//     PlcTask Outputs/GVL_iXlinker.EtherCAT_Master_ERxxxx.Beckhoff_ER2xxx.Beckhoff_ER2xxxEK1122.A_0046_ER2809_0021_0017.Channel_16.Output <-> Channel 16/Output
//     PlcTask Inputs/GVL_iXlinker.EtherCAT_Master_ERxxxx.Beckhoff_ER2xxx.Beckhoff_ER2xxxEK1122.A_0046_ER2809_0021_0017.WcState.WcState <-> WcState/WcState
//     PlcTask Inputs/GVL_iXlinker.EtherCAT_Master_ERxxxx.Beckhoff_ER2xxx.Beckhoff_ER2xxxEK1122.A_0046_ER2809_0021_0017.InfoData.State <-> InfoData/State
//   PLC/PLC Instance <-> EtherCAT Master ERxxxx/Beckhoff ER2xxx/Beckhoff ER2xxxEK1122/A_0047(ER2809-0021-0018)
//     PlcTask Outputs/GVL_iXlinker.EtherCAT_Master_ERxxxx.Beckhoff_ER2xxx.Beckhoff_ER2xxxEK1122.A_0047_ER2809_0021_0018.Channel_1.Output <-> Channel 1/Output
//     PlcTask Outputs/GVL_iXlinker.EtherCAT_Master_ERxxxx.Beckhoff_ER2xxx.Beckhoff_ER2xxxEK1122.A_0047_ER2809_0021_0018.Channel_2.Output <-> Channel 2/Output
//     PlcTask Outputs/GVL_iXlinker.EtherCAT_Master_ERxxxx.Beckhoff_ER2xxx.Beckhoff_ER2xxxEK1122.A_0047_ER2809_0021_0018.Channel_3.Output <-> Channel 3/Output
//     PlcTask Outputs/GVL_iXlinker.EtherCAT_Master_ERxxxx.Beckhoff_ER2xxx.Beckhoff_ER2xxxEK1122.A_0047_ER2809_0021_0018.Channel_4.Output <-> Channel 4/Output
//     PlcTask Outputs/GVL_iXlinker.EtherCAT_Master_ERxxxx.Beckhoff_ER2xxx.Beckhoff_ER2xxxEK1122.A_0047_ER2809_0021_0018.Channel_5.Output <-> Channel 5/Output
//     PlcTask Outputs/GVL_iXlinker.EtherCAT_Master_ERxxxx.Beckhoff_ER2xxx.Beckhoff_ER2xxxEK1122.A_0047_ER2809_0021_0018.Channel_6.Output <-> Channel 6/Output
//     PlcTask Outputs/GVL_iXlinker.EtherCAT_Master_ERxxxx.Beckhoff_ER2xxx.Beckhoff_ER2xxxEK1122.A_0047_ER2809_0021_0018.Channel_7.Output <-> Channel 7/Output
//     PlcTask Outputs/GVL_iXlinker.EtherCAT_Master_ERxxxx.Beckhoff_ER2xxx.Beckhoff_ER2xxxEK1122.A_0047_ER2809_0021_0018.Channel_8.Output <-> Channel 8/Output
//     PlcTask Outputs/GVL_iXlinker.EtherCAT_Master_ERxxxx.Beckhoff_ER2xxx.Beckhoff_ER2xxxEK1122.A_0047_ER2809_0021_0018.Channel_9.Output <-> Channel 9/Output
//     PlcTask Outputs/GVL_iXlinker.EtherCAT_Master_ERxxxx.Beckhoff_ER2xxx.Beckhoff_ER2xxxEK1122.A_0047_ER2809_0021_0018.Channel_10.Output <-> Channel 10/Output
//     PlcTask Outputs/GVL_iXlinker.EtherCAT_Master_ERxxxx.Beckhoff_ER2xxx.Beckhoff_ER2xxxEK1122.A_0047_ER2809_0021_0018.Channel_11.Output <-> Channel 11/Output
//     PlcTask Outputs/GVL_iXlinker.EtherCAT_Master_ERxxxx.Beckhoff_ER2xxx.Beckhoff_ER2xxxEK1122.A_0047_ER2809_0021_0018.Channel_12.Output <-> Channel 12/Output
//     PlcTask Outputs/GVL_iXlinker.EtherCAT_Master_ERxxxx.Beckhoff_ER2xxx.Beckhoff_ER2xxxEK1122.A_0047_ER2809_0021_0018.Channel_13.Output <-> Channel 13/Output
//     PlcTask Outputs/GVL_iXlinker.EtherCAT_Master_ERxxxx.Beckhoff_ER2xxx.Beckhoff_ER2xxxEK1122.A_0047_ER2809_0021_0018.Channel_14.Output <-> Channel 14/Output
//     PlcTask Outputs/GVL_iXlinker.EtherCAT_Master_ERxxxx.Beckhoff_ER2xxx.Beckhoff_ER2xxxEK1122.A_0047_ER2809_0021_0018.Channel_15.Output <-> Channel 15/Output
//     PlcTask Outputs/GVL_iXlinker.EtherCAT_Master_ERxxxx.Beckhoff_ER2xxx.Beckhoff_ER2xxxEK1122.A_0047_ER2809_0021_0018.Channel_16.Output <-> Channel 16/Output
//     PlcTask Inputs/GVL_iXlinker.EtherCAT_Master_ERxxxx.Beckhoff_ER2xxx.Beckhoff_ER2xxxEK1122.A_0047_ER2809_0021_0018.WcState.WcState <-> WcState/WcState
//     PlcTask Inputs/GVL_iXlinker.EtherCAT_Master_ERxxxx.Beckhoff_ER2xxx.Beckhoff_ER2xxxEK1122.A_0047_ER2809_0021_0018.InfoData.State <-> InfoData/State
//   PLC/PLC Instance <-> EtherCAT Master ERxxxx/Beckhoff ER2xxx/Beckhoff ER2xxxEK1122/A_0048(ER2809-0022-0016)
//     PlcTask Outputs/GVL_iXlinker.EtherCAT_Master_ERxxxx.Beckhoff_ER2xxx.Beckhoff_ER2xxxEK1122.A_0048_ER2809_0022_0016.Channel_1.Output <-> Channel 1/Output
//     PlcTask Outputs/GVL_iXlinker.EtherCAT_Master_ERxxxx.Beckhoff_ER2xxx.Beckhoff_ER2xxxEK1122.A_0048_ER2809_0022_0016.Channel_2.Output <-> Channel 2/Output
//     PlcTask Outputs/GVL_iXlinker.EtherCAT_Master_ERxxxx.Beckhoff_ER2xxx.Beckhoff_ER2xxxEK1122.A_0048_ER2809_0022_0016.Channel_3.Output <-> Channel 3/Output
//     PlcTask Outputs/GVL_iXlinker.EtherCAT_Master_ERxxxx.Beckhoff_ER2xxx.Beckhoff_ER2xxxEK1122.A_0048_ER2809_0022_0016.Channel_4.Output <-> Channel 4/Output
//     PlcTask Outputs/GVL_iXlinker.EtherCAT_Master_ERxxxx.Beckhoff_ER2xxx.Beckhoff_ER2xxxEK1122.A_0048_ER2809_0022_0016.Channel_5.Output <-> Channel 5/Output
//     PlcTask Outputs/GVL_iXlinker.EtherCAT_Master_ERxxxx.Beckhoff_ER2xxx.Beckhoff_ER2xxxEK1122.A_0048_ER2809_0022_0016.Channel_6.Output <-> Channel 6/Output
//     PlcTask Outputs/GVL_iXlinker.EtherCAT_Master_ERxxxx.Beckhoff_ER2xxx.Beckhoff_ER2xxxEK1122.A_0048_ER2809_0022_0016.Channel_7.Output <-> Channel 7/Output
//     PlcTask Outputs/GVL_iXlinker.EtherCAT_Master_ERxxxx.Beckhoff_ER2xxx.Beckhoff_ER2xxxEK1122.A_0048_ER2809_0022_0016.Channel_8.Output <-> Channel 8/Output
//     PlcTask Outputs/GVL_iXlinker.EtherCAT_Master_ERxxxx.Beckhoff_ER2xxx.Beckhoff_ER2xxxEK1122.A_0048_ER2809_0022_0016.Channel_9.Output <-> Channel 9/Output
//     PlcTask Outputs/GVL_iXlinker.EtherCAT_Master_ERxxxx.Beckhoff_ER2xxx.Beckhoff_ER2xxxEK1122.A_0048_ER2809_0022_0016.Channel_10.Output <-> Channel 10/Output
//     PlcTask Outputs/GVL_iXlinker.EtherCAT_Master_ERxxxx.Beckhoff_ER2xxx.Beckhoff_ER2xxxEK1122.A_0048_ER2809_0022_0016.Channel_11.Output <-> Channel 11/Output
//     PlcTask Outputs/GVL_iXlinker.EtherCAT_Master_ERxxxx.Beckhoff_ER2xxx.Beckhoff_ER2xxxEK1122.A_0048_ER2809_0022_0016.Channel_12.Output <-> Channel 12/Output
//     PlcTask Outputs/GVL_iXlinker.EtherCAT_Master_ERxxxx.Beckhoff_ER2xxx.Beckhoff_ER2xxxEK1122.A_0048_ER2809_0022_0016.Channel_13.Output <-> Channel 13/Output
//     PlcTask Outputs/GVL_iXlinker.EtherCAT_Master_ERxxxx.Beckhoff_ER2xxx.Beckhoff_ER2xxxEK1122.A_0048_ER2809_0022_0016.Channel_14.Output <-> Channel 14/Output
//     PlcTask Outputs/GVL_iXlinker.EtherCAT_Master_ERxxxx.Beckhoff_ER2xxx.Beckhoff_ER2xxxEK1122.A_0048_ER2809_0022_0016.Channel_15.Output <-> Channel 15/Output
//     PlcTask Outputs/GVL_iXlinker.EtherCAT_Master_ERxxxx.Beckhoff_ER2xxx.Beckhoff_ER2xxxEK1122.A_0048_ER2809_0022_0016.Channel_16.Output <-> Channel 16/Output
//     PlcTask Inputs/GVL_iXlinker.EtherCAT_Master_ERxxxx.Beckhoff_ER2xxx.Beckhoff_ER2xxxEK1122.A_0048_ER2809_0022_0016.WcState.WcState <-> WcState/WcState
//     PlcTask Inputs/GVL_iXlinker.EtherCAT_Master_ERxxxx.Beckhoff_ER2xxx.Beckhoff_ER2xxxEK1122.A_0048_ER2809_0022_0016.InfoData.State <-> InfoData/State
//   PLC/PLC Instance <-> EtherCAT Master ERxxxx/Beckhoff ER2xxx/Beckhoff ER2xxxEK1122/A_0049(ER2809-0022-0017)
//     PlcTask Outputs/GVL_iXlinker.EtherCAT_Master_ERxxxx.Beckhoff_ER2xxx.Beckhoff_ER2xxxEK1122.A_0049_ER2809_0022_0017.Channel_1.Output <-> Channel 1/Output
//     PlcTask Outputs/GVL_iXlinker.EtherCAT_Master_ERxxxx.Beckhoff_ER2xxx.Beckhoff_ER2xxxEK1122.A_0049_ER2809_0022_0017.Channel_2.Output <-> Channel 2/Output
//     PlcTask Outputs/GVL_iXlinker.EtherCAT_Master_ERxxxx.Beckhoff_ER2xxx.Beckhoff_ER2xxxEK1122.A_0049_ER2809_0022_0017.Channel_3.Output <-> Channel 3/Output
//     PlcTask Outputs/GVL_iXlinker.EtherCAT_Master_ERxxxx.Beckhoff_ER2xxx.Beckhoff_ER2xxxEK1122.A_0049_ER2809_0022_0017.Channel_4.Output <-> Channel 4/Output
//     PlcTask Outputs/GVL_iXlinker.EtherCAT_Master_ERxxxx.Beckhoff_ER2xxx.Beckhoff_ER2xxxEK1122.A_0049_ER2809_0022_0017.Channel_5.Output <-> Channel 5/Output
//     PlcTask Outputs/GVL_iXlinker.EtherCAT_Master_ERxxxx.Beckhoff_ER2xxx.Beckhoff_ER2xxxEK1122.A_0049_ER2809_0022_0017.Channel_6.Output <-> Channel 6/Output
//     PlcTask Outputs/GVL_iXlinker.EtherCAT_Master_ERxxxx.Beckhoff_ER2xxx.Beckhoff_ER2xxxEK1122.A_0049_ER2809_0022_0017.Channel_7.Output <-> Channel 7/Output
//     PlcTask Outputs/GVL_iXlinker.EtherCAT_Master_ERxxxx.Beckhoff_ER2xxx.Beckhoff_ER2xxxEK1122.A_0049_ER2809_0022_0017.Channel_8.Output <-> Channel 8/Output
//     PlcTask Outputs/GVL_iXlinker.EtherCAT_Master_ERxxxx.Beckhoff_ER2xxx.Beckhoff_ER2xxxEK1122.A_0049_ER2809_0022_0017.Channel_9.Output <-> Channel 9/Output
//     PlcTask Outputs/GVL_iXlinker.EtherCAT_Master_ERxxxx.Beckhoff_ER2xxx.Beckhoff_ER2xxxEK1122.A_0049_ER2809_0022_0017.Channel_10.Output <-> Channel 10/Output
//     PlcTask Outputs/GVL_iXlinker.EtherCAT_Master_ERxxxx.Beckhoff_ER2xxx.Beckhoff_ER2xxxEK1122.A_0049_ER2809_0022_0017.Channel_11.Output <-> Channel 11/Output
//     PlcTask Outputs/GVL_iXlinker.EtherCAT_Master_ERxxxx.Beckhoff_ER2xxx.Beckhoff_ER2xxxEK1122.A_0049_ER2809_0022_0017.Channel_12.Output <-> Channel 12/Output
//     PlcTask Outputs/GVL_iXlinker.EtherCAT_Master_ERxxxx.Beckhoff_ER2xxx.Beckhoff_ER2xxxEK1122.A_0049_ER2809_0022_0017.Channel_13.Output <-> Channel 13/Output
//     PlcTask Outputs/GVL_iXlinker.EtherCAT_Master_ERxxxx.Beckhoff_ER2xxx.Beckhoff_ER2xxxEK1122.A_0049_ER2809_0022_0017.Channel_14.Output <-> Channel 14/Output
//     PlcTask Outputs/GVL_iXlinker.EtherCAT_Master_ERxxxx.Beckhoff_ER2xxx.Beckhoff_ER2xxxEK1122.A_0049_ER2809_0022_0017.Channel_15.Output <-> Channel 15/Output
//     PlcTask Outputs/GVL_iXlinker.EtherCAT_Master_ERxxxx.Beckhoff_ER2xxx.Beckhoff_ER2xxxEK1122.A_0049_ER2809_0022_0017.Channel_16.Output <-> Channel 16/Output
//     PlcTask Inputs/GVL_iXlinker.EtherCAT_Master_ERxxxx.Beckhoff_ER2xxx.Beckhoff_ER2xxxEK1122.A_0049_ER2809_0022_0017.WcState.WcState <-> WcState/WcState
//     PlcTask Inputs/GVL_iXlinker.EtherCAT_Master_ERxxxx.Beckhoff_ER2xxx.Beckhoff_ER2xxxEK1122.A_0049_ER2809_0022_0017.InfoData.State <-> InfoData/State
//   PLC/PLC Instance <-> EtherCAT Master ERxxxx/Beckhoff ER2xxx/Beckhoff ER2xxxEK1122/A_0050(ER2809-0022-0018)
//     PlcTask Outputs/GVL_iXlinker.EtherCAT_Master_ERxxxx.Beckhoff_ER2xxx.Beckhoff_ER2xxxEK1122.A_0050_ER2809_0022_0018.Channel_1.Output <-> Channel 1/Output
//     PlcTask Outputs/GVL_iXlinker.EtherCAT_Master_ERxxxx.Beckhoff_ER2xxx.Beckhoff_ER2xxxEK1122.A_0050_ER2809_0022_0018.Channel_2.Output <-> Channel 2/Output
//     PlcTask Outputs/GVL_iXlinker.EtherCAT_Master_ERxxxx.Beckhoff_ER2xxx.Beckhoff_ER2xxxEK1122.A_0050_ER2809_0022_0018.Channel_3.Output <-> Channel 3/Output
//     PlcTask Outputs/GVL_iXlinker.EtherCAT_Master_ERxxxx.Beckhoff_ER2xxx.Beckhoff_ER2xxxEK1122.A_0050_ER2809_0022_0018.Channel_4.Output <-> Channel 4/Output
//     PlcTask Outputs/GVL_iXlinker.EtherCAT_Master_ERxxxx.Beckhoff_ER2xxx.Beckhoff_ER2xxxEK1122.A_0050_ER2809_0022_0018.Channel_5.Output <-> Channel 5/Output
//     PlcTask Outputs/GVL_iXlinker.EtherCAT_Master_ERxxxx.Beckhoff_ER2xxx.Beckhoff_ER2xxxEK1122.A_0050_ER2809_0022_0018.Channel_6.Output <-> Channel 6/Output
//     PlcTask Outputs/GVL_iXlinker.EtherCAT_Master_ERxxxx.Beckhoff_ER2xxx.Beckhoff_ER2xxxEK1122.A_0050_ER2809_0022_0018.Channel_7.Output <-> Channel 7/Output
//     PlcTask Outputs/GVL_iXlinker.EtherCAT_Master_ERxxxx.Beckhoff_ER2xxx.Beckhoff_ER2xxxEK1122.A_0050_ER2809_0022_0018.Channel_8.Output <-> Channel 8/Output
//     PlcTask Outputs/GVL_iXlinker.EtherCAT_Master_ERxxxx.Beckhoff_ER2xxx.Beckhoff_ER2xxxEK1122.A_0050_ER2809_0022_0018.Channel_9.Output <-> Channel 9/Output
//     PlcTask Outputs/GVL_iXlinker.EtherCAT_Master_ERxxxx.Beckhoff_ER2xxx.Beckhoff_ER2xxxEK1122.A_0050_ER2809_0022_0018.Channel_10.Output <-> Channel 10/Output
//     PlcTask Outputs/GVL_iXlinker.EtherCAT_Master_ERxxxx.Beckhoff_ER2xxx.Beckhoff_ER2xxxEK1122.A_0050_ER2809_0022_0018.Channel_11.Output <-> Channel 11/Output
//     PlcTask Outputs/GVL_iXlinker.EtherCAT_Master_ERxxxx.Beckhoff_ER2xxx.Beckhoff_ER2xxxEK1122.A_0050_ER2809_0022_0018.Channel_12.Output <-> Channel 12/Output
//     PlcTask Outputs/GVL_iXlinker.EtherCAT_Master_ERxxxx.Beckhoff_ER2xxx.Beckhoff_ER2xxxEK1122.A_0050_ER2809_0022_0018.Channel_13.Output <-> Channel 13/Output
//     PlcTask Outputs/GVL_iXlinker.EtherCAT_Master_ERxxxx.Beckhoff_ER2xxx.Beckhoff_ER2xxxEK1122.A_0050_ER2809_0022_0018.Channel_14.Output <-> Channel 14/Output
//     PlcTask Outputs/GVL_iXlinker.EtherCAT_Master_ERxxxx.Beckhoff_ER2xxx.Beckhoff_ER2xxxEK1122.A_0050_ER2809_0022_0018.Channel_15.Output <-> Channel 15/Output
//     PlcTask Outputs/GVL_iXlinker.EtherCAT_Master_ERxxxx.Beckhoff_ER2xxx.Beckhoff_ER2xxxEK1122.A_0050_ER2809_0022_0018.Channel_16.Output <-> Channel 16/Output
//     PlcTask Inputs/GVL_iXlinker.EtherCAT_Master_ERxxxx.Beckhoff_ER2xxx.Beckhoff_ER2xxxEK1122.A_0050_ER2809_0022_0018.WcState.WcState <-> WcState/WcState
//     PlcTask Inputs/GVL_iXlinker.EtherCAT_Master_ERxxxx.Beckhoff_ER2xxx.Beckhoff_ER2xxxEK1122.A_0050_ER2809_0022_0018.InfoData.State <-> InfoData/State
//   PLC/PLC Instance <-> EtherCAT Master ERxxxx/Beckhoff ER3xxx
//     PlcTask Inputs/GVL_iXlinker.EtherCAT_Master_ERxxxx.Beckhoff_ER3xxx.InfoData.State <-> InfoData/State
//   PLC/PLC Instance <-> EtherCAT Master ERxxxx/Beckhoff ER3xxx/Beckhoff ER3xxxEK1122
//     PlcTask Inputs/GVL_iXlinker.EtherCAT_Master_ERxxxx.Beckhoff_ER3xxx.Beckhoff_ER3xxxEK1122.InfoData.State <-> InfoData/State
//   PLC/PLC Instance <-> EtherCAT Master ERxxxx/Beckhoff ER3xxx/Beckhoff ER3xxxEK1122/Beckhoff ER3xxxsub EK1100
//     PlcTask Inputs/GVL_iXlinker.EtherCAT_Master_ERxxxx.Beckhoff_ER3xxx.Beckhoff_ER3xxxEK1122.Beckhoff_ER3xxxsub_EK1100.InfoData.State <-> InfoData/State
//   PLC/PLC Instance <-> EtherCAT Master ERxxxx/Beckhoff ER3xxx/Beckhoff ER3xxxEK1122/A_0001(ER3174-0002-0016)
//     PlcTask Inputs/GVL_iXlinker.EtherCAT_Master_ERxxxx.Beckhoff_ER3xxx.Beckhoff_ER3xxxEK1122.A_0001_ER3174_0002_0016.AI_Standard_Channel_1.Status/Underrange <-> AI Standard Channel 1/Status/Underrange
//     PlcTask Inputs/GVL_iXlinker.EtherCAT_Master_ERxxxx.Beckhoff_ER3xxx.Beckhoff_ER3xxxEK1122.A_0001_ER3174_0002_0016.AI_Standard_Channel_2.Status/Underrange <-> AI Standard Channel 2/Status/Underrange
//     PlcTask Inputs/GVL_iXlinker.EtherCAT_Master_ERxxxx.Beckhoff_ER3xxx.Beckhoff_ER3xxxEK1122.A_0001_ER3174_0002_0016.AI_Standard_Channel_3.Status/Underrange <-> AI Standard Channel 3/Status/Underrange
//     PlcTask Inputs/GVL_iXlinker.EtherCAT_Master_ERxxxx.Beckhoff_ER3xxx.Beckhoff_ER3xxxEK1122.A_0001_ER3174_0002_0016.AI_Standard_Channel_4.Status/Underrange <-> AI Standard Channel 4/Status/Underrange
//     PlcTask Inputs/GVL_iXlinker.EtherCAT_Master_ERxxxx.Beckhoff_ER3xxx.Beckhoff_ER3xxxEK1122.A_0001_ER3174_0002_0016.AI_Standard_Channel_1.Status/Overrange <-> AI Standard Channel 1/Status/Overrange
//     PlcTask Inputs/GVL_iXlinker.EtherCAT_Master_ERxxxx.Beckhoff_ER3xxx.Beckhoff_ER3xxxEK1122.A_0001_ER3174_0002_0016.AI_Standard_Channel_2.Status/Overrange <-> AI Standard Channel 2/Status/Overrange
//     PlcTask Inputs/GVL_iXlinker.EtherCAT_Master_ERxxxx.Beckhoff_ER3xxx.Beckhoff_ER3xxxEK1122.A_0001_ER3174_0002_0016.AI_Standard_Channel_3.Status/Overrange <-> AI Standard Channel 3/Status/Overrange
//     PlcTask Inputs/GVL_iXlinker.EtherCAT_Master_ERxxxx.Beckhoff_ER3xxx.Beckhoff_ER3xxxEK1122.A_0001_ER3174_0002_0016.AI_Standard_Channel_4.Status/Overrange <-> AI Standard Channel 4/Status/Overrange
//     PlcTask Inputs/GVL_iXlinker.EtherCAT_Master_ERxxxx.Beckhoff_ER3xxx.Beckhoff_ER3xxxEK1122.A_0001_ER3174_0002_0016.AI_Standard_Channel_1.Status/Limit_1 <-> AI Standard Channel 1/Status/Limit 1
//     PlcTask Inputs/GVL_iXlinker.EtherCAT_Master_ERxxxx.Beckhoff_ER3xxx.Beckhoff_ER3xxxEK1122.A_0001_ER3174_0002_0016.AI_Standard_Channel_1.Status/Limit_2 <-> AI Standard Channel 1/Status/Limit 2
//     PlcTask Inputs/GVL_iXlinker.EtherCAT_Master_ERxxxx.Beckhoff_ER3xxx.Beckhoff_ER3xxxEK1122.A_0001_ER3174_0002_0016.AI_Standard_Channel_2.Status/Limit_1 <-> AI Standard Channel 2/Status/Limit 1
//     PlcTask Inputs/GVL_iXlinker.EtherCAT_Master_ERxxxx.Beckhoff_ER3xxx.Beckhoff_ER3xxxEK1122.A_0001_ER3174_0002_0016.AI_Standard_Channel_2.Status/Limit_2 <-> AI Standard Channel 2/Status/Limit 2
//     PlcTask Inputs/GVL_iXlinker.EtherCAT_Master_ERxxxx.Beckhoff_ER3xxx.Beckhoff_ER3xxxEK1122.A_0001_ER3174_0002_0016.AI_Standard_Channel_3.Status/Limit_1 <-> AI Standard Channel 3/Status/Limit 1
//     PlcTask Inputs/GVL_iXlinker.EtherCAT_Master_ERxxxx.Beckhoff_ER3xxx.Beckhoff_ER3xxxEK1122.A_0001_ER3174_0002_0016.AI_Standard_Channel_3.Status/Limit_2 <-> AI Standard Channel 3/Status/Limit 2
//     PlcTask Inputs/GVL_iXlinker.EtherCAT_Master_ERxxxx.Beckhoff_ER3xxx.Beckhoff_ER3xxxEK1122.A_0001_ER3174_0002_0016.AI_Standard_Channel_4.Status/Limit_1 <-> AI Standard Channel 4/Status/Limit 1
//     PlcTask Inputs/GVL_iXlinker.EtherCAT_Master_ERxxxx.Beckhoff_ER3xxx.Beckhoff_ER3xxxEK1122.A_0001_ER3174_0002_0016.AI_Standard_Channel_4.Status/Limit_2 <-> AI Standard Channel 4/Status/Limit 2
//     PlcTask Inputs/GVL_iXlinker.EtherCAT_Master_ERxxxx.Beckhoff_ER3xxx.Beckhoff_ER3xxxEK1122.A_0001_ER3174_0002_0016.AI_Standard_Channel_1.Status/Error <-> AI Standard Channel 1/Status/Error
//     PlcTask Inputs/GVL_iXlinker.EtherCAT_Master_ERxxxx.Beckhoff_ER3xxx.Beckhoff_ER3xxxEK1122.A_0001_ER3174_0002_0016.AI_Standard_Channel_2.Status/Error <-> AI Standard Channel 2/Status/Error
//     PlcTask Inputs/GVL_iXlinker.EtherCAT_Master_ERxxxx.Beckhoff_ER3xxx.Beckhoff_ER3xxxEK1122.A_0001_ER3174_0002_0016.AI_Standard_Channel_3.Status/Error <-> AI Standard Channel 3/Status/Error
//     PlcTask Inputs/GVL_iXlinker.EtherCAT_Master_ERxxxx.Beckhoff_ER3xxx.Beckhoff_ER3xxxEK1122.A_0001_ER3174_0002_0016.AI_Standard_Channel_4.Status/Error <-> AI Standard Channel 4/Status/Error
//     PlcTask Inputs/GVL_iXlinker.EtherCAT_Master_ERxxxx.Beckhoff_ER3xxx.Beckhoff_ER3xxxEK1122.A_0001_ER3174_0002_0016.AI_Standard_Channel_1.Status/Sync_error <-> AI Standard Channel 1/Status/Sync error
//     PlcTask Inputs/GVL_iXlinker.EtherCAT_Master_ERxxxx.Beckhoff_ER3xxx.Beckhoff_ER3xxxEK1122.A_0001_ER3174_0002_0016.AI_Standard_Channel_2.Status/Sync_error <-> AI Standard Channel 2/Status/Sync error
//     PlcTask Inputs/GVL_iXlinker.EtherCAT_Master_ERxxxx.Beckhoff_ER3xxx.Beckhoff_ER3xxxEK1122.A_0001_ER3174_0002_0016.AI_Standard_Channel_3.Status/Sync_error <-> AI Standard Channel 3/Status/Sync error
//     PlcTask Inputs/GVL_iXlinker.EtherCAT_Master_ERxxxx.Beckhoff_ER3xxx.Beckhoff_ER3xxxEK1122.A_0001_ER3174_0002_0016.AI_Standard_Channel_4.Status/Sync_error <-> AI Standard Channel 4/Status/Sync error
//     PlcTask Inputs/GVL_iXlinker.EtherCAT_Master_ERxxxx.Beckhoff_ER3xxx.Beckhoff_ER3xxxEK1122.A_0001_ER3174_0002_0016.AI_Standard_Channel_1.Status/TxPDO_State <-> AI Standard Channel 1/Status/TxPDO State
//     PlcTask Inputs/GVL_iXlinker.EtherCAT_Master_ERxxxx.Beckhoff_ER3xxx.Beckhoff_ER3xxxEK1122.A_0001_ER3174_0002_0016.AI_Standard_Channel_2.Status/TxPDO_State <-> AI Standard Channel 2/Status/TxPDO State
//     PlcTask Inputs/GVL_iXlinker.EtherCAT_Master_ERxxxx.Beckhoff_ER3xxx.Beckhoff_ER3xxxEK1122.A_0001_ER3174_0002_0016.AI_Standard_Channel_3.Status/TxPDO_State <-> AI Standard Channel 3/Status/TxPDO State
//     PlcTask Inputs/GVL_iXlinker.EtherCAT_Master_ERxxxx.Beckhoff_ER3xxx.Beckhoff_ER3xxxEK1122.A_0001_ER3174_0002_0016.AI_Standard_Channel_4.Status/TxPDO_State <-> AI Standard Channel 4/Status/TxPDO State
//     PlcTask Inputs/GVL_iXlinker.EtherCAT_Master_ERxxxx.Beckhoff_ER3xxx.Beckhoff_ER3xxxEK1122.A_0001_ER3174_0002_0016.AI_Standard_Channel_1.Status/TxPDO_Toggle <-> AI Standard Channel 1/Status/TxPDO Toggle
//     PlcTask Inputs/GVL_iXlinker.EtherCAT_Master_ERxxxx.Beckhoff_ER3xxx.Beckhoff_ER3xxxEK1122.A_0001_ER3174_0002_0016.AI_Standard_Channel_2.Status/TxPDO_Toggle <-> AI Standard Channel 2/Status/TxPDO Toggle
//     PlcTask Inputs/GVL_iXlinker.EtherCAT_Master_ERxxxx.Beckhoff_ER3xxx.Beckhoff_ER3xxxEK1122.A_0001_ER3174_0002_0016.AI_Standard_Channel_3.Status/TxPDO_Toggle <-> AI Standard Channel 3/Status/TxPDO Toggle
//     PlcTask Inputs/GVL_iXlinker.EtherCAT_Master_ERxxxx.Beckhoff_ER3xxx.Beckhoff_ER3xxxEK1122.A_0001_ER3174_0002_0016.AI_Standard_Channel_4.Status/TxPDO_Toggle <-> AI Standard Channel 4/Status/TxPDO Toggle
//     PlcTask Inputs/GVL_iXlinker.EtherCAT_Master_ERxxxx.Beckhoff_ER3xxx.Beckhoff_ER3xxxEK1122.A_0001_ER3174_0002_0016.AI_Standard_Channel_1.Value <-> AI Standard Channel 1/Value
//     PlcTask Inputs/GVL_iXlinker.EtherCAT_Master_ERxxxx.Beckhoff_ER3xxx.Beckhoff_ER3xxxEK1122.A_0001_ER3174_0002_0016.AI_Standard_Channel_2.Value <-> AI Standard Channel 2/Value
//     PlcTask Inputs/GVL_iXlinker.EtherCAT_Master_ERxxxx.Beckhoff_ER3xxx.Beckhoff_ER3xxxEK1122.A_0001_ER3174_0002_0016.AI_Standard_Channel_3.Value <-> AI Standard Channel 3/Value
//     PlcTask Inputs/GVL_iXlinker.EtherCAT_Master_ERxxxx.Beckhoff_ER3xxx.Beckhoff_ER3xxxEK1122.A_0001_ER3174_0002_0016.AI_Standard_Channel_4.Value <-> AI Standard Channel 4/Value
//     PlcTask Inputs/GVL_iXlinker.EtherCAT_Master_ERxxxx.Beckhoff_ER3xxx.Beckhoff_ER3xxxEK1122.A_0001_ER3174_0002_0016.WcState.WcState <-> WcState/WcState
//     PlcTask Inputs/GVL_iXlinker.EtherCAT_Master_ERxxxx.Beckhoff_ER3xxx.Beckhoff_ER3xxxEK1122.A_0001_ER3174_0002_0016.WcState.InputToggle <-> WcState/InputToggle
//     PlcTask Inputs/GVL_iXlinker.EtherCAT_Master_ERxxxx.Beckhoff_ER3xxx.Beckhoff_ER3xxxEK1122.A_0001_ER3174_0002_0016.InfoData.AdsAddr <-> InfoData/AdsAddr
//     PlcTask Inputs/GVL_iXlinker.EtherCAT_Master_ERxxxx.Beckhoff_ER3xxx.Beckhoff_ER3xxxEK1122.A_0001_ER3174_0002_0016.InfoData.State <-> InfoData/State
//   PLC/PLC Instance <-> EtherCAT Master ERxxxx/Beckhoff ER3xxx/Beckhoff ER3xxxEK1122/A_0002(ER3174-0002-0022)
//     PlcTask Inputs/GVL_iXlinker.EtherCAT_Master_ERxxxx.Beckhoff_ER3xxx.Beckhoff_ER3xxxEK1122.A_0002_ER3174_0002_0022.AI_Standard_Channel_1.Status/Underrange <-> AI Standard Channel 1/Status/Underrange
//     PlcTask Inputs/GVL_iXlinker.EtherCAT_Master_ERxxxx.Beckhoff_ER3xxx.Beckhoff_ER3xxxEK1122.A_0002_ER3174_0002_0022.AI_Standard_Channel_2.Status/Underrange <-> AI Standard Channel 2/Status/Underrange
//     PlcTask Inputs/GVL_iXlinker.EtherCAT_Master_ERxxxx.Beckhoff_ER3xxx.Beckhoff_ER3xxxEK1122.A_0002_ER3174_0002_0022.AI_Standard_Channel_3.Status/Underrange <-> AI Standard Channel 3/Status/Underrange
//     PlcTask Inputs/GVL_iXlinker.EtherCAT_Master_ERxxxx.Beckhoff_ER3xxx.Beckhoff_ER3xxxEK1122.A_0002_ER3174_0002_0022.AI_Standard_Channel_4.Status/Underrange <-> AI Standard Channel 4/Status/Underrange
//     PlcTask Inputs/GVL_iXlinker.EtherCAT_Master_ERxxxx.Beckhoff_ER3xxx.Beckhoff_ER3xxxEK1122.A_0002_ER3174_0002_0022.AI_Standard_Channel_1.Status/Overrange <-> AI Standard Channel 1/Status/Overrange
//     PlcTask Inputs/GVL_iXlinker.EtherCAT_Master_ERxxxx.Beckhoff_ER3xxx.Beckhoff_ER3xxxEK1122.A_0002_ER3174_0002_0022.AI_Standard_Channel_2.Status/Overrange <-> AI Standard Channel 2/Status/Overrange
//     PlcTask Inputs/GVL_iXlinker.EtherCAT_Master_ERxxxx.Beckhoff_ER3xxx.Beckhoff_ER3xxxEK1122.A_0002_ER3174_0002_0022.AI_Standard_Channel_3.Status/Overrange <-> AI Standard Channel 3/Status/Overrange
//     PlcTask Inputs/GVL_iXlinker.EtherCAT_Master_ERxxxx.Beckhoff_ER3xxx.Beckhoff_ER3xxxEK1122.A_0002_ER3174_0002_0022.AI_Standard_Channel_4.Status/Overrange <-> AI Standard Channel 4/Status/Overrange
//     PlcTask Inputs/GVL_iXlinker.EtherCAT_Master_ERxxxx.Beckhoff_ER3xxx.Beckhoff_ER3xxxEK1122.A_0002_ER3174_0002_0022.AI_Standard_Channel_1.Status/Limit_1 <-> AI Standard Channel 1/Status/Limit 1
//     PlcTask Inputs/GVL_iXlinker.EtherCAT_Master_ERxxxx.Beckhoff_ER3xxx.Beckhoff_ER3xxxEK1122.A_0002_ER3174_0002_0022.AI_Standard_Channel_1.Status/Limit_2 <-> AI Standard Channel 1/Status/Limit 2
//     PlcTask Inputs/GVL_iXlinker.EtherCAT_Master_ERxxxx.Beckhoff_ER3xxx.Beckhoff_ER3xxxEK1122.A_0002_ER3174_0002_0022.AI_Standard_Channel_2.Status/Limit_1 <-> AI Standard Channel 2/Status/Limit 1
//     PlcTask Inputs/GVL_iXlinker.EtherCAT_Master_ERxxxx.Beckhoff_ER3xxx.Beckhoff_ER3xxxEK1122.A_0002_ER3174_0002_0022.AI_Standard_Channel_2.Status/Limit_2 <-> AI Standard Channel 2/Status/Limit 2
//     PlcTask Inputs/GVL_iXlinker.EtherCAT_Master_ERxxxx.Beckhoff_ER3xxx.Beckhoff_ER3xxxEK1122.A_0002_ER3174_0002_0022.AI_Standard_Channel_3.Status/Limit_1 <-> AI Standard Channel 3/Status/Limit 1
//     PlcTask Inputs/GVL_iXlinker.EtherCAT_Master_ERxxxx.Beckhoff_ER3xxx.Beckhoff_ER3xxxEK1122.A_0002_ER3174_0002_0022.AI_Standard_Channel_3.Status/Limit_2 <-> AI Standard Channel 3/Status/Limit 2
//     PlcTask Inputs/GVL_iXlinker.EtherCAT_Master_ERxxxx.Beckhoff_ER3xxx.Beckhoff_ER3xxxEK1122.A_0002_ER3174_0002_0022.AI_Standard_Channel_4.Status/Limit_1 <-> AI Standard Channel 4/Status/Limit 1
//     PlcTask Inputs/GVL_iXlinker.EtherCAT_Master_ERxxxx.Beckhoff_ER3xxx.Beckhoff_ER3xxxEK1122.A_0002_ER3174_0002_0022.AI_Standard_Channel_4.Status/Limit_2 <-> AI Standard Channel 4/Status/Limit 2
//     PlcTask Inputs/GVL_iXlinker.EtherCAT_Master_ERxxxx.Beckhoff_ER3xxx.Beckhoff_ER3xxxEK1122.A_0002_ER3174_0002_0022.AI_Standard_Channel_1.Status/Error <-> AI Standard Channel 1/Status/Error
//     PlcTask Inputs/GVL_iXlinker.EtherCAT_Master_ERxxxx.Beckhoff_ER3xxx.Beckhoff_ER3xxxEK1122.A_0002_ER3174_0002_0022.AI_Standard_Channel_2.Status/Error <-> AI Standard Channel 2/Status/Error
//     PlcTask Inputs/GVL_iXlinker.EtherCAT_Master_ERxxxx.Beckhoff_ER3xxx.Beckhoff_ER3xxxEK1122.A_0002_ER3174_0002_0022.AI_Standard_Channel_3.Status/Error <-> AI Standard Channel 3/Status/Error
//     PlcTask Inputs/GVL_iXlinker.EtherCAT_Master_ERxxxx.Beckhoff_ER3xxx.Beckhoff_ER3xxxEK1122.A_0002_ER3174_0002_0022.AI_Standard_Channel_4.Status/Error <-> AI Standard Channel 4/Status/Error
//     PlcTask Inputs/GVL_iXlinker.EtherCAT_Master_ERxxxx.Beckhoff_ER3xxx.Beckhoff_ER3xxxEK1122.A_0002_ER3174_0002_0022.AI_Standard_Channel_1.Status/Sync_error <-> AI Standard Channel 1/Status/Sync error
//     PlcTask Inputs/GVL_iXlinker.EtherCAT_Master_ERxxxx.Beckhoff_ER3xxx.Beckhoff_ER3xxxEK1122.A_0002_ER3174_0002_0022.AI_Standard_Channel_2.Status/Sync_error <-> AI Standard Channel 2/Status/Sync error
//     PlcTask Inputs/GVL_iXlinker.EtherCAT_Master_ERxxxx.Beckhoff_ER3xxx.Beckhoff_ER3xxxEK1122.A_0002_ER3174_0002_0022.AI_Standard_Channel_3.Status/Sync_error <-> AI Standard Channel 3/Status/Sync error
//     PlcTask Inputs/GVL_iXlinker.EtherCAT_Master_ERxxxx.Beckhoff_ER3xxx.Beckhoff_ER3xxxEK1122.A_0002_ER3174_0002_0022.AI_Standard_Channel_4.Status/Sync_error <-> AI Standard Channel 4/Status/Sync error
//     PlcTask Inputs/GVL_iXlinker.EtherCAT_Master_ERxxxx.Beckhoff_ER3xxx.Beckhoff_ER3xxxEK1122.A_0002_ER3174_0002_0022.AI_Standard_Channel_1.Status/TxPDO_State <-> AI Standard Channel 1/Status/TxPDO State
//     PlcTask Inputs/GVL_iXlinker.EtherCAT_Master_ERxxxx.Beckhoff_ER3xxx.Beckhoff_ER3xxxEK1122.A_0002_ER3174_0002_0022.AI_Standard_Channel_2.Status/TxPDO_State <-> AI Standard Channel 2/Status/TxPDO State
//     PlcTask Inputs/GVL_iXlinker.EtherCAT_Master_ERxxxx.Beckhoff_ER3xxx.Beckhoff_ER3xxxEK1122.A_0002_ER3174_0002_0022.AI_Standard_Channel_3.Status/TxPDO_State <-> AI Standard Channel 3/Status/TxPDO State
//     PlcTask Inputs/GVL_iXlinker.EtherCAT_Master_ERxxxx.Beckhoff_ER3xxx.Beckhoff_ER3xxxEK1122.A_0002_ER3174_0002_0022.AI_Standard_Channel_4.Status/TxPDO_State <-> AI Standard Channel 4/Status/TxPDO State
//     PlcTask Inputs/GVL_iXlinker.EtherCAT_Master_ERxxxx.Beckhoff_ER3xxx.Beckhoff_ER3xxxEK1122.A_0002_ER3174_0002_0022.AI_Standard_Channel_1.Status/TxPDO_Toggle <-> AI Standard Channel 1/Status/TxPDO Toggle
//     PlcTask Inputs/GVL_iXlinker.EtherCAT_Master_ERxxxx.Beckhoff_ER3xxx.Beckhoff_ER3xxxEK1122.A_0002_ER3174_0002_0022.AI_Standard_Channel_2.Status/TxPDO_Toggle <-> AI Standard Channel 2/Status/TxPDO Toggle
//     PlcTask Inputs/GVL_iXlinker.EtherCAT_Master_ERxxxx.Beckhoff_ER3xxx.Beckhoff_ER3xxxEK1122.A_0002_ER3174_0002_0022.AI_Standard_Channel_3.Status/TxPDO_Toggle <-> AI Standard Channel 3/Status/TxPDO Toggle
//     PlcTask Inputs/GVL_iXlinker.EtherCAT_Master_ERxxxx.Beckhoff_ER3xxx.Beckhoff_ER3xxxEK1122.A_0002_ER3174_0002_0022.AI_Standard_Channel_4.Status/TxPDO_Toggle <-> AI Standard Channel 4/Status/TxPDO Toggle
//     PlcTask Inputs/GVL_iXlinker.EtherCAT_Master_ERxxxx.Beckhoff_ER3xxx.Beckhoff_ER3xxxEK1122.A_0002_ER3174_0002_0022.AI_Standard_Channel_1.Value <-> AI Standard Channel 1/Value
//     PlcTask Inputs/GVL_iXlinker.EtherCAT_Master_ERxxxx.Beckhoff_ER3xxx.Beckhoff_ER3xxxEK1122.A_0002_ER3174_0002_0022.AI_Standard_Channel_2.Value <-> AI Standard Channel 2/Value
//     PlcTask Inputs/GVL_iXlinker.EtherCAT_Master_ERxxxx.Beckhoff_ER3xxx.Beckhoff_ER3xxxEK1122.A_0002_ER3174_0002_0022.AI_Standard_Channel_3.Value <-> AI Standard Channel 3/Value
//     PlcTask Inputs/GVL_iXlinker.EtherCAT_Master_ERxxxx.Beckhoff_ER3xxx.Beckhoff_ER3xxxEK1122.A_0002_ER3174_0002_0022.AI_Standard_Channel_4.Value <-> AI Standard Channel 4/Value
//     PlcTask Inputs/GVL_iXlinker.EtherCAT_Master_ERxxxx.Beckhoff_ER3xxx.Beckhoff_ER3xxxEK1122.A_0002_ER3174_0002_0022.WcState.WcState <-> WcState/WcState
//     PlcTask Inputs/GVL_iXlinker.EtherCAT_Master_ERxxxx.Beckhoff_ER3xxx.Beckhoff_ER3xxxEK1122.A_0002_ER3174_0002_0022.WcState.InputToggle <-> WcState/InputToggle
//     PlcTask Inputs/GVL_iXlinker.EtherCAT_Master_ERxxxx.Beckhoff_ER3xxx.Beckhoff_ER3xxxEK1122.A_0002_ER3174_0002_0022.InfoData.AdsAddr <-> InfoData/AdsAddr
//     PlcTask Inputs/GVL_iXlinker.EtherCAT_Master_ERxxxx.Beckhoff_ER3xxx.Beckhoff_ER3xxxEK1122.A_0002_ER3174_0002_0022.InfoData.State <-> InfoData/State
//   PLC/PLC Instance <-> EtherCAT Master ERxxxx/Beckhoff ER3xxx/Beckhoff ER3xxxEK1122/A_0003(ER3174-0002-0023)
//     PlcTask Inputs/GVL_iXlinker.EtherCAT_Master_ERxxxx.Beckhoff_ER3xxx.Beckhoff_ER3xxxEK1122.A_0003_ER3174_0002_0023.AI_Standard_Channel_1.Status/Underrange <-> AI Standard Channel 1/Status/Underrange
//     PlcTask Inputs/GVL_iXlinker.EtherCAT_Master_ERxxxx.Beckhoff_ER3xxx.Beckhoff_ER3xxxEK1122.A_0003_ER3174_0002_0023.AI_Standard_Channel_2.Status/Underrange <-> AI Standard Channel 2/Status/Underrange
//     PlcTask Inputs/GVL_iXlinker.EtherCAT_Master_ERxxxx.Beckhoff_ER3xxx.Beckhoff_ER3xxxEK1122.A_0003_ER3174_0002_0023.AI_Standard_Channel_3.Status/Underrange <-> AI Standard Channel 3/Status/Underrange
//     PlcTask Inputs/GVL_iXlinker.EtherCAT_Master_ERxxxx.Beckhoff_ER3xxx.Beckhoff_ER3xxxEK1122.A_0003_ER3174_0002_0023.AI_Standard_Channel_4.Status/Underrange <-> AI Standard Channel 4/Status/Underrange
//     PlcTask Inputs/GVL_iXlinker.EtherCAT_Master_ERxxxx.Beckhoff_ER3xxx.Beckhoff_ER3xxxEK1122.A_0003_ER3174_0002_0023.AI_Standard_Channel_1.Status/Overrange <-> AI Standard Channel 1/Status/Overrange
//     PlcTask Inputs/GVL_iXlinker.EtherCAT_Master_ERxxxx.Beckhoff_ER3xxx.Beckhoff_ER3xxxEK1122.A_0003_ER3174_0002_0023.AI_Standard_Channel_2.Status/Overrange <-> AI Standard Channel 2/Status/Overrange
//     PlcTask Inputs/GVL_iXlinker.EtherCAT_Master_ERxxxx.Beckhoff_ER3xxx.Beckhoff_ER3xxxEK1122.A_0003_ER3174_0002_0023.AI_Standard_Channel_3.Status/Overrange <-> AI Standard Channel 3/Status/Overrange
//     PlcTask Inputs/GVL_iXlinker.EtherCAT_Master_ERxxxx.Beckhoff_ER3xxx.Beckhoff_ER3xxxEK1122.A_0003_ER3174_0002_0023.AI_Standard_Channel_4.Status/Overrange <-> AI Standard Channel 4/Status/Overrange
//     PlcTask Inputs/GVL_iXlinker.EtherCAT_Master_ERxxxx.Beckhoff_ER3xxx.Beckhoff_ER3xxxEK1122.A_0003_ER3174_0002_0023.AI_Standard_Channel_1.Status/Limit_1 <-> AI Standard Channel 1/Status/Limit 1
//     PlcTask Inputs/GVL_iXlinker.EtherCAT_Master_ERxxxx.Beckhoff_ER3xxx.Beckhoff_ER3xxxEK1122.A_0003_ER3174_0002_0023.AI_Standard_Channel_1.Status/Limit_2 <-> AI Standard Channel 1/Status/Limit 2
//     PlcTask Inputs/GVL_iXlinker.EtherCAT_Master_ERxxxx.Beckhoff_ER3xxx.Beckhoff_ER3xxxEK1122.A_0003_ER3174_0002_0023.AI_Standard_Channel_2.Status/Limit_1 <-> AI Standard Channel 2/Status/Limit 1
//     PlcTask Inputs/GVL_iXlinker.EtherCAT_Master_ERxxxx.Beckhoff_ER3xxx.Beckhoff_ER3xxxEK1122.A_0003_ER3174_0002_0023.AI_Standard_Channel_2.Status/Limit_2 <-> AI Standard Channel 2/Status/Limit 2
//     PlcTask Inputs/GVL_iXlinker.EtherCAT_Master_ERxxxx.Beckhoff_ER3xxx.Beckhoff_ER3xxxEK1122.A_0003_ER3174_0002_0023.AI_Standard_Channel_3.Status/Limit_1 <-> AI Standard Channel 3/Status/Limit 1
//     PlcTask Inputs/GVL_iXlinker.EtherCAT_Master_ERxxxx.Beckhoff_ER3xxx.Beckhoff_ER3xxxEK1122.A_0003_ER3174_0002_0023.AI_Standard_Channel_3.Status/Limit_2 <-> AI Standard Channel 3/Status/Limit 2
//     PlcTask Inputs/GVL_iXlinker.EtherCAT_Master_ERxxxx.Beckhoff_ER3xxx.Beckhoff_ER3xxxEK1122.A_0003_ER3174_0002_0023.AI_Standard_Channel_4.Status/Limit_1 <-> AI Standard Channel 4/Status/Limit 1
//     PlcTask Inputs/GVL_iXlinker.EtherCAT_Master_ERxxxx.Beckhoff_ER3xxx.Beckhoff_ER3xxxEK1122.A_0003_ER3174_0002_0023.AI_Standard_Channel_4.Status/Limit_2 <-> AI Standard Channel 4/Status/Limit 2
//     PlcTask Inputs/GVL_iXlinker.EtherCAT_Master_ERxxxx.Beckhoff_ER3xxx.Beckhoff_ER3xxxEK1122.A_0003_ER3174_0002_0023.AI_Standard_Channel_1.Status/Error <-> AI Standard Channel 1/Status/Error
//     PlcTask Inputs/GVL_iXlinker.EtherCAT_Master_ERxxxx.Beckhoff_ER3xxx.Beckhoff_ER3xxxEK1122.A_0003_ER3174_0002_0023.AI_Standard_Channel_2.Status/Error <-> AI Standard Channel 2/Status/Error
//     PlcTask Inputs/GVL_iXlinker.EtherCAT_Master_ERxxxx.Beckhoff_ER3xxx.Beckhoff_ER3xxxEK1122.A_0003_ER3174_0002_0023.AI_Standard_Channel_3.Status/Error <-> AI Standard Channel 3/Status/Error
//     PlcTask Inputs/GVL_iXlinker.EtherCAT_Master_ERxxxx.Beckhoff_ER3xxx.Beckhoff_ER3xxxEK1122.A_0003_ER3174_0002_0023.AI_Standard_Channel_4.Status/Error <-> AI Standard Channel 4/Status/Error
//     PlcTask Inputs/GVL_iXlinker.EtherCAT_Master_ERxxxx.Beckhoff_ER3xxx.Beckhoff_ER3xxxEK1122.A_0003_ER3174_0002_0023.AI_Standard_Channel_1.Status/Sync_error <-> AI Standard Channel 1/Status/Sync error
//     PlcTask Inputs/GVL_iXlinker.EtherCAT_Master_ERxxxx.Beckhoff_ER3xxx.Beckhoff_ER3xxxEK1122.A_0003_ER3174_0002_0023.AI_Standard_Channel_2.Status/Sync_error <-> AI Standard Channel 2/Status/Sync error
//     PlcTask Inputs/GVL_iXlinker.EtherCAT_Master_ERxxxx.Beckhoff_ER3xxx.Beckhoff_ER3xxxEK1122.A_0003_ER3174_0002_0023.AI_Standard_Channel_3.Status/Sync_error <-> AI Standard Channel 3/Status/Sync error
//     PlcTask Inputs/GVL_iXlinker.EtherCAT_Master_ERxxxx.Beckhoff_ER3xxx.Beckhoff_ER3xxxEK1122.A_0003_ER3174_0002_0023.AI_Standard_Channel_4.Status/Sync_error <-> AI Standard Channel 4/Status/Sync error
//     PlcTask Inputs/GVL_iXlinker.EtherCAT_Master_ERxxxx.Beckhoff_ER3xxx.Beckhoff_ER3xxxEK1122.A_0003_ER3174_0002_0023.AI_Standard_Channel_1.Status/TxPDO_State <-> AI Standard Channel 1/Status/TxPDO State
//     PlcTask Inputs/GVL_iXlinker.EtherCAT_Master_ERxxxx.Beckhoff_ER3xxx.Beckhoff_ER3xxxEK1122.A_0003_ER3174_0002_0023.AI_Standard_Channel_2.Status/TxPDO_State <-> AI Standard Channel 2/Status/TxPDO State
//     PlcTask Inputs/GVL_iXlinker.EtherCAT_Master_ERxxxx.Beckhoff_ER3xxx.Beckhoff_ER3xxxEK1122.A_0003_ER3174_0002_0023.AI_Standard_Channel_3.Status/TxPDO_State <-> AI Standard Channel 3/Status/TxPDO State
//     PlcTask Inputs/GVL_iXlinker.EtherCAT_Master_ERxxxx.Beckhoff_ER3xxx.Beckhoff_ER3xxxEK1122.A_0003_ER3174_0002_0023.AI_Standard_Channel_4.Status/TxPDO_State <-> AI Standard Channel 4/Status/TxPDO State
//     PlcTask Inputs/GVL_iXlinker.EtherCAT_Master_ERxxxx.Beckhoff_ER3xxx.Beckhoff_ER3xxxEK1122.A_0003_ER3174_0002_0023.AI_Standard_Channel_1.Status/TxPDO_Toggle <-> AI Standard Channel 1/Status/TxPDO Toggle
//     PlcTask Inputs/GVL_iXlinker.EtherCAT_Master_ERxxxx.Beckhoff_ER3xxx.Beckhoff_ER3xxxEK1122.A_0003_ER3174_0002_0023.AI_Standard_Channel_2.Status/TxPDO_Toggle <-> AI Standard Channel 2/Status/TxPDO Toggle
//     PlcTask Inputs/GVL_iXlinker.EtherCAT_Master_ERxxxx.Beckhoff_ER3xxx.Beckhoff_ER3xxxEK1122.A_0003_ER3174_0002_0023.AI_Standard_Channel_3.Status/TxPDO_Toggle <-> AI Standard Channel 3/Status/TxPDO Toggle
//     PlcTask Inputs/GVL_iXlinker.EtherCAT_Master_ERxxxx.Beckhoff_ER3xxx.Beckhoff_ER3xxxEK1122.A_0003_ER3174_0002_0023.AI_Standard_Channel_4.Status/TxPDO_Toggle <-> AI Standard Channel 4/Status/TxPDO Toggle
//     PlcTask Inputs/GVL_iXlinker.EtherCAT_Master_ERxxxx.Beckhoff_ER3xxx.Beckhoff_ER3xxxEK1122.A_0003_ER3174_0002_0023.AI_Standard_Channel_1.Value <-> AI Standard Channel 1/Value
//     PlcTask Inputs/GVL_iXlinker.EtherCAT_Master_ERxxxx.Beckhoff_ER3xxx.Beckhoff_ER3xxxEK1122.A_0003_ER3174_0002_0023.AI_Standard_Channel_2.Value <-> AI Standard Channel 2/Value
//     PlcTask Inputs/GVL_iXlinker.EtherCAT_Master_ERxxxx.Beckhoff_ER3xxx.Beckhoff_ER3xxxEK1122.A_0003_ER3174_0002_0023.AI_Standard_Channel_3.Value <-> AI Standard Channel 3/Value
//     PlcTask Inputs/GVL_iXlinker.EtherCAT_Master_ERxxxx.Beckhoff_ER3xxx.Beckhoff_ER3xxxEK1122.A_0003_ER3174_0002_0023.AI_Standard_Channel_4.Value <-> AI Standard Channel 4/Value
//     PlcTask Inputs/GVL_iXlinker.EtherCAT_Master_ERxxxx.Beckhoff_ER3xxx.Beckhoff_ER3xxxEK1122.A_0003_ER3174_0002_0023.WcState.WcState <-> WcState/WcState
//     PlcTask Inputs/GVL_iXlinker.EtherCAT_Master_ERxxxx.Beckhoff_ER3xxx.Beckhoff_ER3xxxEK1122.A_0003_ER3174_0002_0023.WcState.InputToggle <-> WcState/InputToggle
//     PlcTask Inputs/GVL_iXlinker.EtherCAT_Master_ERxxxx.Beckhoff_ER3xxx.Beckhoff_ER3xxxEK1122.A_0003_ER3174_0002_0023.InfoData.AdsAddr <-> InfoData/AdsAddr
//     PlcTask Inputs/GVL_iXlinker.EtherCAT_Master_ERxxxx.Beckhoff_ER3xxx.Beckhoff_ER3xxxEK1122.A_0003_ER3174_0002_0023.InfoData.State <-> InfoData/State
//   PLC/PLC Instance <-> EtherCAT Master ERxxxx/Beckhoff ER3xxx/Beckhoff ER3xxxEK1122/A_0004(ER3184-0002-0019)
//     PlcTask Inputs/GVL_iXlinker.EtherCAT_Master_ERxxxx.Beckhoff_ER3xxx.Beckhoff_ER3xxxEK1122.A_0004_ER3184_0002_0019.AI_Standard_Channel_1.Status/Underrange <-> AI Standard Channel 1/Status/Underrange
//     PlcTask Inputs/GVL_iXlinker.EtherCAT_Master_ERxxxx.Beckhoff_ER3xxx.Beckhoff_ER3xxxEK1122.A_0004_ER3184_0002_0019.AI_Standard_Channel_2.Status/Underrange <-> AI Standard Channel 2/Status/Underrange
//     PlcTask Inputs/GVL_iXlinker.EtherCAT_Master_ERxxxx.Beckhoff_ER3xxx.Beckhoff_ER3xxxEK1122.A_0004_ER3184_0002_0019.AI_Standard_Channel_3.Status/Underrange <-> AI Standard Channel 3/Status/Underrange
//     PlcTask Inputs/GVL_iXlinker.EtherCAT_Master_ERxxxx.Beckhoff_ER3xxx.Beckhoff_ER3xxxEK1122.A_0004_ER3184_0002_0019.AI_Standard_Channel_4.Status/Underrange <-> AI Standard Channel 4/Status/Underrange
//     PlcTask Inputs/GVL_iXlinker.EtherCAT_Master_ERxxxx.Beckhoff_ER3xxx.Beckhoff_ER3xxxEK1122.A_0004_ER3184_0002_0019.AI_Standard_Channel_1.Status/Overrange <-> AI Standard Channel 1/Status/Overrange
//     PlcTask Inputs/GVL_iXlinker.EtherCAT_Master_ERxxxx.Beckhoff_ER3xxx.Beckhoff_ER3xxxEK1122.A_0004_ER3184_0002_0019.AI_Standard_Channel_2.Status/Overrange <-> AI Standard Channel 2/Status/Overrange
//     PlcTask Inputs/GVL_iXlinker.EtherCAT_Master_ERxxxx.Beckhoff_ER3xxx.Beckhoff_ER3xxxEK1122.A_0004_ER3184_0002_0019.AI_Standard_Channel_3.Status/Overrange <-> AI Standard Channel 3/Status/Overrange
//     PlcTask Inputs/GVL_iXlinker.EtherCAT_Master_ERxxxx.Beckhoff_ER3xxx.Beckhoff_ER3xxxEK1122.A_0004_ER3184_0002_0019.AI_Standard_Channel_4.Status/Overrange <-> AI Standard Channel 4/Status/Overrange
//     PlcTask Inputs/GVL_iXlinker.EtherCAT_Master_ERxxxx.Beckhoff_ER3xxx.Beckhoff_ER3xxxEK1122.A_0004_ER3184_0002_0019.AI_Standard_Channel_1.Status/Limit_1 <-> AI Standard Channel 1/Status/Limit 1
//     PlcTask Inputs/GVL_iXlinker.EtherCAT_Master_ERxxxx.Beckhoff_ER3xxx.Beckhoff_ER3xxxEK1122.A_0004_ER3184_0002_0019.AI_Standard_Channel_1.Status/Limit_2 <-> AI Standard Channel 1/Status/Limit 2
//     PlcTask Inputs/GVL_iXlinker.EtherCAT_Master_ERxxxx.Beckhoff_ER3xxx.Beckhoff_ER3xxxEK1122.A_0004_ER3184_0002_0019.AI_Standard_Channel_2.Status/Limit_1 <-> AI Standard Channel 2/Status/Limit 1
//     PlcTask Inputs/GVL_iXlinker.EtherCAT_Master_ERxxxx.Beckhoff_ER3xxx.Beckhoff_ER3xxxEK1122.A_0004_ER3184_0002_0019.AI_Standard_Channel_2.Status/Limit_2 <-> AI Standard Channel 2/Status/Limit 2
//     PlcTask Inputs/GVL_iXlinker.EtherCAT_Master_ERxxxx.Beckhoff_ER3xxx.Beckhoff_ER3xxxEK1122.A_0004_ER3184_0002_0019.AI_Standard_Channel_3.Status/Limit_1 <-> AI Standard Channel 3/Status/Limit 1
//     PlcTask Inputs/GVL_iXlinker.EtherCAT_Master_ERxxxx.Beckhoff_ER3xxx.Beckhoff_ER3xxxEK1122.A_0004_ER3184_0002_0019.AI_Standard_Channel_3.Status/Limit_2 <-> AI Standard Channel 3/Status/Limit 2
//     PlcTask Inputs/GVL_iXlinker.EtherCAT_Master_ERxxxx.Beckhoff_ER3xxx.Beckhoff_ER3xxxEK1122.A_0004_ER3184_0002_0019.AI_Standard_Channel_4.Status/Limit_1 <-> AI Standard Channel 4/Status/Limit 1
//     PlcTask Inputs/GVL_iXlinker.EtherCAT_Master_ERxxxx.Beckhoff_ER3xxx.Beckhoff_ER3xxxEK1122.A_0004_ER3184_0002_0019.AI_Standard_Channel_4.Status/Limit_2 <-> AI Standard Channel 4/Status/Limit 2
//     PlcTask Inputs/GVL_iXlinker.EtherCAT_Master_ERxxxx.Beckhoff_ER3xxx.Beckhoff_ER3xxxEK1122.A_0004_ER3184_0002_0019.AI_Standard_Channel_1.Status/Error <-> AI Standard Channel 1/Status/Error
//     PlcTask Inputs/GVL_iXlinker.EtherCAT_Master_ERxxxx.Beckhoff_ER3xxx.Beckhoff_ER3xxxEK1122.A_0004_ER3184_0002_0019.AI_Standard_Channel_2.Status/Error <-> AI Standard Channel 2/Status/Error
//     PlcTask Inputs/GVL_iXlinker.EtherCAT_Master_ERxxxx.Beckhoff_ER3xxx.Beckhoff_ER3xxxEK1122.A_0004_ER3184_0002_0019.AI_Standard_Channel_3.Status/Error <-> AI Standard Channel 3/Status/Error
//     PlcTask Inputs/GVL_iXlinker.EtherCAT_Master_ERxxxx.Beckhoff_ER3xxx.Beckhoff_ER3xxxEK1122.A_0004_ER3184_0002_0019.AI_Standard_Channel_4.Status/Error <-> AI Standard Channel 4/Status/Error
//     PlcTask Inputs/GVL_iXlinker.EtherCAT_Master_ERxxxx.Beckhoff_ER3xxx.Beckhoff_ER3xxxEK1122.A_0004_ER3184_0002_0019.AI_Standard_Channel_1.Status/Sync_error <-> AI Standard Channel 1/Status/Sync error
//     PlcTask Inputs/GVL_iXlinker.EtherCAT_Master_ERxxxx.Beckhoff_ER3xxx.Beckhoff_ER3xxxEK1122.A_0004_ER3184_0002_0019.AI_Standard_Channel_2.Status/Sync_error <-> AI Standard Channel 2/Status/Sync error
//     PlcTask Inputs/GVL_iXlinker.EtherCAT_Master_ERxxxx.Beckhoff_ER3xxx.Beckhoff_ER3xxxEK1122.A_0004_ER3184_0002_0019.AI_Standard_Channel_3.Status/Sync_error <-> AI Standard Channel 3/Status/Sync error
//     PlcTask Inputs/GVL_iXlinker.EtherCAT_Master_ERxxxx.Beckhoff_ER3xxx.Beckhoff_ER3xxxEK1122.A_0004_ER3184_0002_0019.AI_Standard_Channel_4.Status/Sync_error <-> AI Standard Channel 4/Status/Sync error
//     PlcTask Inputs/GVL_iXlinker.EtherCAT_Master_ERxxxx.Beckhoff_ER3xxx.Beckhoff_ER3xxxEK1122.A_0004_ER3184_0002_0019.AI_Standard_Channel_1.Status/TxPDO_State <-> AI Standard Channel 1/Status/TxPDO State
//     PlcTask Inputs/GVL_iXlinker.EtherCAT_Master_ERxxxx.Beckhoff_ER3xxx.Beckhoff_ER3xxxEK1122.A_0004_ER3184_0002_0019.AI_Standard_Channel_2.Status/TxPDO_State <-> AI Standard Channel 2/Status/TxPDO State
//     PlcTask Inputs/GVL_iXlinker.EtherCAT_Master_ERxxxx.Beckhoff_ER3xxx.Beckhoff_ER3xxxEK1122.A_0004_ER3184_0002_0019.AI_Standard_Channel_3.Status/TxPDO_State <-> AI Standard Channel 3/Status/TxPDO State
//     PlcTask Inputs/GVL_iXlinker.EtherCAT_Master_ERxxxx.Beckhoff_ER3xxx.Beckhoff_ER3xxxEK1122.A_0004_ER3184_0002_0019.AI_Standard_Channel_4.Status/TxPDO_State <-> AI Standard Channel 4/Status/TxPDO State
//     PlcTask Inputs/GVL_iXlinker.EtherCAT_Master_ERxxxx.Beckhoff_ER3xxx.Beckhoff_ER3xxxEK1122.A_0004_ER3184_0002_0019.AI_Standard_Channel_1.Status/TxPDO_Toggle <-> AI Standard Channel 1/Status/TxPDO Toggle
//     PlcTask Inputs/GVL_iXlinker.EtherCAT_Master_ERxxxx.Beckhoff_ER3xxx.Beckhoff_ER3xxxEK1122.A_0004_ER3184_0002_0019.AI_Standard_Channel_2.Status/TxPDO_Toggle <-> AI Standard Channel 2/Status/TxPDO Toggle
//     PlcTask Inputs/GVL_iXlinker.EtherCAT_Master_ERxxxx.Beckhoff_ER3xxx.Beckhoff_ER3xxxEK1122.A_0004_ER3184_0002_0019.AI_Standard_Channel_3.Status/TxPDO_Toggle <-> AI Standard Channel 3/Status/TxPDO Toggle
//     PlcTask Inputs/GVL_iXlinker.EtherCAT_Master_ERxxxx.Beckhoff_ER3xxx.Beckhoff_ER3xxxEK1122.A_0004_ER3184_0002_0019.AI_Standard_Channel_4.Status/TxPDO_Toggle <-> AI Standard Channel 4/Status/TxPDO Toggle
//     PlcTask Inputs/GVL_iXlinker.EtherCAT_Master_ERxxxx.Beckhoff_ER3xxx.Beckhoff_ER3xxxEK1122.A_0004_ER3184_0002_0019.AI_Standard_Channel_1.Value <-> AI Standard Channel 1/Value
//     PlcTask Inputs/GVL_iXlinker.EtherCAT_Master_ERxxxx.Beckhoff_ER3xxx.Beckhoff_ER3xxxEK1122.A_0004_ER3184_0002_0019.AI_Standard_Channel_2.Value <-> AI Standard Channel 2/Value
//     PlcTask Inputs/GVL_iXlinker.EtherCAT_Master_ERxxxx.Beckhoff_ER3xxx.Beckhoff_ER3xxxEK1122.A_0004_ER3184_0002_0019.AI_Standard_Channel_3.Value <-> AI Standard Channel 3/Value
//     PlcTask Inputs/GVL_iXlinker.EtherCAT_Master_ERxxxx.Beckhoff_ER3xxx.Beckhoff_ER3xxxEK1122.A_0004_ER3184_0002_0019.AI_Standard_Channel_4.Value <-> AI Standard Channel 4/Value
//     PlcTask Inputs/GVL_iXlinker.EtherCAT_Master_ERxxxx.Beckhoff_ER3xxx.Beckhoff_ER3xxxEK1122.A_0004_ER3184_0002_0019.WcState.WcState <-> WcState/WcState
//     PlcTask Inputs/GVL_iXlinker.EtherCAT_Master_ERxxxx.Beckhoff_ER3xxx.Beckhoff_ER3xxxEK1122.A_0004_ER3184_0002_0019.WcState.InputToggle <-> WcState/InputToggle
//     PlcTask Inputs/GVL_iXlinker.EtherCAT_Master_ERxxxx.Beckhoff_ER3xxx.Beckhoff_ER3xxxEK1122.A_0004_ER3184_0002_0019.InfoData.AdsAddr <-> InfoData/AdsAddr
//     PlcTask Inputs/GVL_iXlinker.EtherCAT_Master_ERxxxx.Beckhoff_ER3xxx.Beckhoff_ER3xxxEK1122.A_0004_ER3184_0002_0019.InfoData.State <-> InfoData/State
//   PLC/PLC Instance <-> EtherCAT Master ERxxxx/Beckhoff ER3xxx/Beckhoff ER3xxxEK1122/A_0005(ER3184-0002-0020)
//     PlcTask Inputs/GVL_iXlinker.EtherCAT_Master_ERxxxx.Beckhoff_ER3xxx.Beckhoff_ER3xxxEK1122.A_0005_ER3184_0002_0020.AI_Standard_Channel_1.Status/Underrange <-> AI Standard Channel 1/Status/Underrange
//     PlcTask Inputs/GVL_iXlinker.EtherCAT_Master_ERxxxx.Beckhoff_ER3xxx.Beckhoff_ER3xxxEK1122.A_0005_ER3184_0002_0020.AI_Standard_Channel_2.Status/Underrange <-> AI Standard Channel 2/Status/Underrange
//     PlcTask Inputs/GVL_iXlinker.EtherCAT_Master_ERxxxx.Beckhoff_ER3xxx.Beckhoff_ER3xxxEK1122.A_0005_ER3184_0002_0020.AI_Standard_Channel_3.Status/Underrange <-> AI Standard Channel 3/Status/Underrange
//     PlcTask Inputs/GVL_iXlinker.EtherCAT_Master_ERxxxx.Beckhoff_ER3xxx.Beckhoff_ER3xxxEK1122.A_0005_ER3184_0002_0020.AI_Standard_Channel_4.Status/Underrange <-> AI Standard Channel 4/Status/Underrange
//     PlcTask Inputs/GVL_iXlinker.EtherCAT_Master_ERxxxx.Beckhoff_ER3xxx.Beckhoff_ER3xxxEK1122.A_0005_ER3184_0002_0020.AI_Standard_Channel_1.Status/Overrange <-> AI Standard Channel 1/Status/Overrange
//     PlcTask Inputs/GVL_iXlinker.EtherCAT_Master_ERxxxx.Beckhoff_ER3xxx.Beckhoff_ER3xxxEK1122.A_0005_ER3184_0002_0020.AI_Standard_Channel_2.Status/Overrange <-> AI Standard Channel 2/Status/Overrange
//     PlcTask Inputs/GVL_iXlinker.EtherCAT_Master_ERxxxx.Beckhoff_ER3xxx.Beckhoff_ER3xxxEK1122.A_0005_ER3184_0002_0020.AI_Standard_Channel_3.Status/Overrange <-> AI Standard Channel 3/Status/Overrange
//     PlcTask Inputs/GVL_iXlinker.EtherCAT_Master_ERxxxx.Beckhoff_ER3xxx.Beckhoff_ER3xxxEK1122.A_0005_ER3184_0002_0020.AI_Standard_Channel_4.Status/Overrange <-> AI Standard Channel 4/Status/Overrange
//     PlcTask Inputs/GVL_iXlinker.EtherCAT_Master_ERxxxx.Beckhoff_ER3xxx.Beckhoff_ER3xxxEK1122.A_0005_ER3184_0002_0020.AI_Standard_Channel_1.Status/Limit_1 <-> AI Standard Channel 1/Status/Limit 1
//     PlcTask Inputs/GVL_iXlinker.EtherCAT_Master_ERxxxx.Beckhoff_ER3xxx.Beckhoff_ER3xxxEK1122.A_0005_ER3184_0002_0020.AI_Standard_Channel_1.Status/Limit_2 <-> AI Standard Channel 1/Status/Limit 2
//     PlcTask Inputs/GVL_iXlinker.EtherCAT_Master_ERxxxx.Beckhoff_ER3xxx.Beckhoff_ER3xxxEK1122.A_0005_ER3184_0002_0020.AI_Standard_Channel_2.Status/Limit_1 <-> AI Standard Channel 2/Status/Limit 1
//     PlcTask Inputs/GVL_iXlinker.EtherCAT_Master_ERxxxx.Beckhoff_ER3xxx.Beckhoff_ER3xxxEK1122.A_0005_ER3184_0002_0020.AI_Standard_Channel_2.Status/Limit_2 <-> AI Standard Channel 2/Status/Limit 2
//     PlcTask Inputs/GVL_iXlinker.EtherCAT_Master_ERxxxx.Beckhoff_ER3xxx.Beckhoff_ER3xxxEK1122.A_0005_ER3184_0002_0020.AI_Standard_Channel_3.Status/Limit_1 <-> AI Standard Channel 3/Status/Limit 1
//     PlcTask Inputs/GVL_iXlinker.EtherCAT_Master_ERxxxx.Beckhoff_ER3xxx.Beckhoff_ER3xxxEK1122.A_0005_ER3184_0002_0020.AI_Standard_Channel_3.Status/Limit_2 <-> AI Standard Channel 3/Status/Limit 2
//     PlcTask Inputs/GVL_iXlinker.EtherCAT_Master_ERxxxx.Beckhoff_ER3xxx.Beckhoff_ER3xxxEK1122.A_0005_ER3184_0002_0020.AI_Standard_Channel_4.Status/Limit_1 <-> AI Standard Channel 4/Status/Limit 1
//     PlcTask Inputs/GVL_iXlinker.EtherCAT_Master_ERxxxx.Beckhoff_ER3xxx.Beckhoff_ER3xxxEK1122.A_0005_ER3184_0002_0020.AI_Standard_Channel_4.Status/Limit_2 <-> AI Standard Channel 4/Status/Limit 2
//     PlcTask Inputs/GVL_iXlinker.EtherCAT_Master_ERxxxx.Beckhoff_ER3xxx.Beckhoff_ER3xxxEK1122.A_0005_ER3184_0002_0020.AI_Standard_Channel_1.Status/Error <-> AI Standard Channel 1/Status/Error
//     PlcTask Inputs/GVL_iXlinker.EtherCAT_Master_ERxxxx.Beckhoff_ER3xxx.Beckhoff_ER3xxxEK1122.A_0005_ER3184_0002_0020.AI_Standard_Channel_2.Status/Error <-> AI Standard Channel 2/Status/Error
//     PlcTask Inputs/GVL_iXlinker.EtherCAT_Master_ERxxxx.Beckhoff_ER3xxx.Beckhoff_ER3xxxEK1122.A_0005_ER3184_0002_0020.AI_Standard_Channel_3.Status/Error <-> AI Standard Channel 3/Status/Error
//     PlcTask Inputs/GVL_iXlinker.EtherCAT_Master_ERxxxx.Beckhoff_ER3xxx.Beckhoff_ER3xxxEK1122.A_0005_ER3184_0002_0020.AI_Standard_Channel_4.Status/Error <-> AI Standard Channel 4/Status/Error
//     PlcTask Inputs/GVL_iXlinker.EtherCAT_Master_ERxxxx.Beckhoff_ER3xxx.Beckhoff_ER3xxxEK1122.A_0005_ER3184_0002_0020.AI_Standard_Channel_1.Status/Sync_error <-> AI Standard Channel 1/Status/Sync error
//     PlcTask Inputs/GVL_iXlinker.EtherCAT_Master_ERxxxx.Beckhoff_ER3xxx.Beckhoff_ER3xxxEK1122.A_0005_ER3184_0002_0020.AI_Standard_Channel_2.Status/Sync_error <-> AI Standard Channel 2/Status/Sync error
//     PlcTask Inputs/GVL_iXlinker.EtherCAT_Master_ERxxxx.Beckhoff_ER3xxx.Beckhoff_ER3xxxEK1122.A_0005_ER3184_0002_0020.AI_Standard_Channel_3.Status/Sync_error <-> AI Standard Channel 3/Status/Sync error
//     PlcTask Inputs/GVL_iXlinker.EtherCAT_Master_ERxxxx.Beckhoff_ER3xxx.Beckhoff_ER3xxxEK1122.A_0005_ER3184_0002_0020.AI_Standard_Channel_4.Status/Sync_error <-> AI Standard Channel 4/Status/Sync error
//     PlcTask Inputs/GVL_iXlinker.EtherCAT_Master_ERxxxx.Beckhoff_ER3xxx.Beckhoff_ER3xxxEK1122.A_0005_ER3184_0002_0020.AI_Standard_Channel_1.Status/TxPDO_State <-> AI Standard Channel 1/Status/TxPDO State
//     PlcTask Inputs/GVL_iXlinker.EtherCAT_Master_ERxxxx.Beckhoff_ER3xxx.Beckhoff_ER3xxxEK1122.A_0005_ER3184_0002_0020.AI_Standard_Channel_2.Status/TxPDO_State <-> AI Standard Channel 2/Status/TxPDO State
//     PlcTask Inputs/GVL_iXlinker.EtherCAT_Master_ERxxxx.Beckhoff_ER3xxx.Beckhoff_ER3xxxEK1122.A_0005_ER3184_0002_0020.AI_Standard_Channel_3.Status/TxPDO_State <-> AI Standard Channel 3/Status/TxPDO State
//     PlcTask Inputs/GVL_iXlinker.EtherCAT_Master_ERxxxx.Beckhoff_ER3xxx.Beckhoff_ER3xxxEK1122.A_0005_ER3184_0002_0020.AI_Standard_Channel_4.Status/TxPDO_State <-> AI Standard Channel 4/Status/TxPDO State
//     PlcTask Inputs/GVL_iXlinker.EtherCAT_Master_ERxxxx.Beckhoff_ER3xxx.Beckhoff_ER3xxxEK1122.A_0005_ER3184_0002_0020.AI_Standard_Channel_1.Status/TxPDO_Toggle <-> AI Standard Channel 1/Status/TxPDO Toggle
//     PlcTask Inputs/GVL_iXlinker.EtherCAT_Master_ERxxxx.Beckhoff_ER3xxx.Beckhoff_ER3xxxEK1122.A_0005_ER3184_0002_0020.AI_Standard_Channel_2.Status/TxPDO_Toggle <-> AI Standard Channel 2/Status/TxPDO Toggle
//     PlcTask Inputs/GVL_iXlinker.EtherCAT_Master_ERxxxx.Beckhoff_ER3xxx.Beckhoff_ER3xxxEK1122.A_0005_ER3184_0002_0020.AI_Standard_Channel_3.Status/TxPDO_Toggle <-> AI Standard Channel 3/Status/TxPDO Toggle
//     PlcTask Inputs/GVL_iXlinker.EtherCAT_Master_ERxxxx.Beckhoff_ER3xxx.Beckhoff_ER3xxxEK1122.A_0005_ER3184_0002_0020.AI_Standard_Channel_4.Status/TxPDO_Toggle <-> AI Standard Channel 4/Status/TxPDO Toggle
//     PlcTask Inputs/GVL_iXlinker.EtherCAT_Master_ERxxxx.Beckhoff_ER3xxx.Beckhoff_ER3xxxEK1122.A_0005_ER3184_0002_0020.AI_Standard_Channel_1.Value <-> AI Standard Channel 1/Value
//     PlcTask Inputs/GVL_iXlinker.EtherCAT_Master_ERxxxx.Beckhoff_ER3xxx.Beckhoff_ER3xxxEK1122.A_0005_ER3184_0002_0020.AI_Standard_Channel_2.Value <-> AI Standard Channel 2/Value
//     PlcTask Inputs/GVL_iXlinker.EtherCAT_Master_ERxxxx.Beckhoff_ER3xxx.Beckhoff_ER3xxxEK1122.A_0005_ER3184_0002_0020.AI_Standard_Channel_3.Value <-> AI Standard Channel 3/Value
//     PlcTask Inputs/GVL_iXlinker.EtherCAT_Master_ERxxxx.Beckhoff_ER3xxx.Beckhoff_ER3xxxEK1122.A_0005_ER3184_0002_0020.AI_Standard_Channel_4.Value <-> AI Standard Channel 4/Value
//     PlcTask Inputs/GVL_iXlinker.EtherCAT_Master_ERxxxx.Beckhoff_ER3xxx.Beckhoff_ER3xxxEK1122.A_0005_ER3184_0002_0020.WcState.WcState <-> WcState/WcState
//     PlcTask Inputs/GVL_iXlinker.EtherCAT_Master_ERxxxx.Beckhoff_ER3xxx.Beckhoff_ER3xxxEK1122.A_0005_ER3184_0002_0020.WcState.InputToggle <-> WcState/InputToggle
//     PlcTask Inputs/GVL_iXlinker.EtherCAT_Master_ERxxxx.Beckhoff_ER3xxx.Beckhoff_ER3xxxEK1122.A_0005_ER3184_0002_0020.InfoData.AdsAddr <-> InfoData/AdsAddr
//     PlcTask Inputs/GVL_iXlinker.EtherCAT_Master_ERxxxx.Beckhoff_ER3xxx.Beckhoff_ER3xxxEK1122.A_0005_ER3184_0002_0020.InfoData.State <-> InfoData/State
//   PLC/PLC Instance <-> EtherCAT Master ERxxxx/Beckhoff ER3xxx/Beckhoff ER3xxxEK1122/A_0006(ER3184-0002-0021)
//     PlcTask Inputs/GVL_iXlinker.EtherCAT_Master_ERxxxx.Beckhoff_ER3xxx.Beckhoff_ER3xxxEK1122.A_0006_ER3184_0002_0021.AI_Standard_Channel_1.Status/Underrange <-> AI Standard Channel 1/Status/Underrange
//     PlcTask Inputs/GVL_iXlinker.EtherCAT_Master_ERxxxx.Beckhoff_ER3xxx.Beckhoff_ER3xxxEK1122.A_0006_ER3184_0002_0021.AI_Standard_Channel_2.Status/Underrange <-> AI Standard Channel 2/Status/Underrange
//     PlcTask Inputs/GVL_iXlinker.EtherCAT_Master_ERxxxx.Beckhoff_ER3xxx.Beckhoff_ER3xxxEK1122.A_0006_ER3184_0002_0021.AI_Standard_Channel_3.Status/Underrange <-> AI Standard Channel 3/Status/Underrange
//     PlcTask Inputs/GVL_iXlinker.EtherCAT_Master_ERxxxx.Beckhoff_ER3xxx.Beckhoff_ER3xxxEK1122.A_0006_ER3184_0002_0021.AI_Standard_Channel_4.Status/Underrange <-> AI Standard Channel 4/Status/Underrange
//     PlcTask Inputs/GVL_iXlinker.EtherCAT_Master_ERxxxx.Beckhoff_ER3xxx.Beckhoff_ER3xxxEK1122.A_0006_ER3184_0002_0021.AI_Standard_Channel_1.Status/Overrange <-> AI Standard Channel 1/Status/Overrange
//     PlcTask Inputs/GVL_iXlinker.EtherCAT_Master_ERxxxx.Beckhoff_ER3xxx.Beckhoff_ER3xxxEK1122.A_0006_ER3184_0002_0021.AI_Standard_Channel_2.Status/Overrange <-> AI Standard Channel 2/Status/Overrange
//     PlcTask Inputs/GVL_iXlinker.EtherCAT_Master_ERxxxx.Beckhoff_ER3xxx.Beckhoff_ER3xxxEK1122.A_0006_ER3184_0002_0021.AI_Standard_Channel_3.Status/Overrange <-> AI Standard Channel 3/Status/Overrange
//     PlcTask Inputs/GVL_iXlinker.EtherCAT_Master_ERxxxx.Beckhoff_ER3xxx.Beckhoff_ER3xxxEK1122.A_0006_ER3184_0002_0021.AI_Standard_Channel_4.Status/Overrange <-> AI Standard Channel 4/Status/Overrange
//     PlcTask Inputs/GVL_iXlinker.EtherCAT_Master_ERxxxx.Beckhoff_ER3xxx.Beckhoff_ER3xxxEK1122.A_0006_ER3184_0002_0021.AI_Standard_Channel_1.Status/Limit_1 <-> AI Standard Channel 1/Status/Limit 1
//     PlcTask Inputs/GVL_iXlinker.EtherCAT_Master_ERxxxx.Beckhoff_ER3xxx.Beckhoff_ER3xxxEK1122.A_0006_ER3184_0002_0021.AI_Standard_Channel_1.Status/Limit_2 <-> AI Standard Channel 1/Status/Limit 2
//     PlcTask Inputs/GVL_iXlinker.EtherCAT_Master_ERxxxx.Beckhoff_ER3xxx.Beckhoff_ER3xxxEK1122.A_0006_ER3184_0002_0021.AI_Standard_Channel_2.Status/Limit_1 <-> AI Standard Channel 2/Status/Limit 1
//     PlcTask Inputs/GVL_iXlinker.EtherCAT_Master_ERxxxx.Beckhoff_ER3xxx.Beckhoff_ER3xxxEK1122.A_0006_ER3184_0002_0021.AI_Standard_Channel_2.Status/Limit_2 <-> AI Standard Channel 2/Status/Limit 2
//     PlcTask Inputs/GVL_iXlinker.EtherCAT_Master_ERxxxx.Beckhoff_ER3xxx.Beckhoff_ER3xxxEK1122.A_0006_ER3184_0002_0021.AI_Standard_Channel_3.Status/Limit_1 <-> AI Standard Channel 3/Status/Limit 1
//     PlcTask Inputs/GVL_iXlinker.EtherCAT_Master_ERxxxx.Beckhoff_ER3xxx.Beckhoff_ER3xxxEK1122.A_0006_ER3184_0002_0021.AI_Standard_Channel_3.Status/Limit_2 <-> AI Standard Channel 3/Status/Limit 2
//     PlcTask Inputs/GVL_iXlinker.EtherCAT_Master_ERxxxx.Beckhoff_ER3xxx.Beckhoff_ER3xxxEK1122.A_0006_ER3184_0002_0021.AI_Standard_Channel_4.Status/Limit_1 <-> AI Standard Channel 4/Status/Limit 1
//     PlcTask Inputs/GVL_iXlinker.EtherCAT_Master_ERxxxx.Beckhoff_ER3xxx.Beckhoff_ER3xxxEK1122.A_0006_ER3184_0002_0021.AI_Standard_Channel_4.Status/Limit_2 <-> AI Standard Channel 4/Status/Limit 2
//     PlcTask Inputs/GVL_iXlinker.EtherCAT_Master_ERxxxx.Beckhoff_ER3xxx.Beckhoff_ER3xxxEK1122.A_0006_ER3184_0002_0021.AI_Standard_Channel_1.Status/Error <-> AI Standard Channel 1/Status/Error
//     PlcTask Inputs/GVL_iXlinker.EtherCAT_Master_ERxxxx.Beckhoff_ER3xxx.Beckhoff_ER3xxxEK1122.A_0006_ER3184_0002_0021.AI_Standard_Channel_2.Status/Error <-> AI Standard Channel 2/Status/Error
//     PlcTask Inputs/GVL_iXlinker.EtherCAT_Master_ERxxxx.Beckhoff_ER3xxx.Beckhoff_ER3xxxEK1122.A_0006_ER3184_0002_0021.AI_Standard_Channel_3.Status/Error <-> AI Standard Channel 3/Status/Error
//     PlcTask Inputs/GVL_iXlinker.EtherCAT_Master_ERxxxx.Beckhoff_ER3xxx.Beckhoff_ER3xxxEK1122.A_0006_ER3184_0002_0021.AI_Standard_Channel_4.Status/Error <-> AI Standard Channel 4/Status/Error
//     PlcTask Inputs/GVL_iXlinker.EtherCAT_Master_ERxxxx.Beckhoff_ER3xxx.Beckhoff_ER3xxxEK1122.A_0006_ER3184_0002_0021.AI_Standard_Channel_1.Status/Sync_error <-> AI Standard Channel 1/Status/Sync error
//     PlcTask Inputs/GVL_iXlinker.EtherCAT_Master_ERxxxx.Beckhoff_ER3xxx.Beckhoff_ER3xxxEK1122.A_0006_ER3184_0002_0021.AI_Standard_Channel_2.Status/Sync_error <-> AI Standard Channel 2/Status/Sync error
//     PlcTask Inputs/GVL_iXlinker.EtherCAT_Master_ERxxxx.Beckhoff_ER3xxx.Beckhoff_ER3xxxEK1122.A_0006_ER3184_0002_0021.AI_Standard_Channel_3.Status/Sync_error <-> AI Standard Channel 3/Status/Sync error
//     PlcTask Inputs/GVL_iXlinker.EtherCAT_Master_ERxxxx.Beckhoff_ER3xxx.Beckhoff_ER3xxxEK1122.A_0006_ER3184_0002_0021.AI_Standard_Channel_4.Status/Sync_error <-> AI Standard Channel 4/Status/Sync error
//     PlcTask Inputs/GVL_iXlinker.EtherCAT_Master_ERxxxx.Beckhoff_ER3xxx.Beckhoff_ER3xxxEK1122.A_0006_ER3184_0002_0021.AI_Standard_Channel_1.Status/TxPDO_State <-> AI Standard Channel 1/Status/TxPDO State
//     PlcTask Inputs/GVL_iXlinker.EtherCAT_Master_ERxxxx.Beckhoff_ER3xxx.Beckhoff_ER3xxxEK1122.A_0006_ER3184_0002_0021.AI_Standard_Channel_2.Status/TxPDO_State <-> AI Standard Channel 2/Status/TxPDO State
//     PlcTask Inputs/GVL_iXlinker.EtherCAT_Master_ERxxxx.Beckhoff_ER3xxx.Beckhoff_ER3xxxEK1122.A_0006_ER3184_0002_0021.AI_Standard_Channel_3.Status/TxPDO_State <-> AI Standard Channel 3/Status/TxPDO State
//     PlcTask Inputs/GVL_iXlinker.EtherCAT_Master_ERxxxx.Beckhoff_ER3xxx.Beckhoff_ER3xxxEK1122.A_0006_ER3184_0002_0021.AI_Standard_Channel_4.Status/TxPDO_State <-> AI Standard Channel 4/Status/TxPDO State
//     PlcTask Inputs/GVL_iXlinker.EtherCAT_Master_ERxxxx.Beckhoff_ER3xxx.Beckhoff_ER3xxxEK1122.A_0006_ER3184_0002_0021.AI_Standard_Channel_1.Status/TxPDO_Toggle <-> AI Standard Channel 1/Status/TxPDO Toggle
//     PlcTask Inputs/GVL_iXlinker.EtherCAT_Master_ERxxxx.Beckhoff_ER3xxx.Beckhoff_ER3xxxEK1122.A_0006_ER3184_0002_0021.AI_Standard_Channel_2.Status/TxPDO_Toggle <-> AI Standard Channel 2/Status/TxPDO Toggle
//     PlcTask Inputs/GVL_iXlinker.EtherCAT_Master_ERxxxx.Beckhoff_ER3xxx.Beckhoff_ER3xxxEK1122.A_0006_ER3184_0002_0021.AI_Standard_Channel_3.Status/TxPDO_Toggle <-> AI Standard Channel 3/Status/TxPDO Toggle
//     PlcTask Inputs/GVL_iXlinker.EtherCAT_Master_ERxxxx.Beckhoff_ER3xxx.Beckhoff_ER3xxxEK1122.A_0006_ER3184_0002_0021.AI_Standard_Channel_4.Status/TxPDO_Toggle <-> AI Standard Channel 4/Status/TxPDO Toggle
//     PlcTask Inputs/GVL_iXlinker.EtherCAT_Master_ERxxxx.Beckhoff_ER3xxx.Beckhoff_ER3xxxEK1122.A_0006_ER3184_0002_0021.AI_Standard_Channel_1.Value <-> AI Standard Channel 1/Value
//     PlcTask Inputs/GVL_iXlinker.EtherCAT_Master_ERxxxx.Beckhoff_ER3xxx.Beckhoff_ER3xxxEK1122.A_0006_ER3184_0002_0021.AI_Standard_Channel_2.Value <-> AI Standard Channel 2/Value
//     PlcTask Inputs/GVL_iXlinker.EtherCAT_Master_ERxxxx.Beckhoff_ER3xxx.Beckhoff_ER3xxxEK1122.A_0006_ER3184_0002_0021.AI_Standard_Channel_3.Value <-> AI Standard Channel 3/Value
//     PlcTask Inputs/GVL_iXlinker.EtherCAT_Master_ERxxxx.Beckhoff_ER3xxx.Beckhoff_ER3xxxEK1122.A_0006_ER3184_0002_0021.AI_Standard_Channel_4.Value <-> AI Standard Channel 4/Value
//     PlcTask Inputs/GVL_iXlinker.EtherCAT_Master_ERxxxx.Beckhoff_ER3xxx.Beckhoff_ER3xxxEK1122.A_0006_ER3184_0002_0021.WcState.WcState <-> WcState/WcState
//     PlcTask Inputs/GVL_iXlinker.EtherCAT_Master_ERxxxx.Beckhoff_ER3xxx.Beckhoff_ER3xxxEK1122.A_0006_ER3184_0002_0021.WcState.InputToggle <-> WcState/InputToggle
//     PlcTask Inputs/GVL_iXlinker.EtherCAT_Master_ERxxxx.Beckhoff_ER3xxx.Beckhoff_ER3xxxEK1122.A_0006_ER3184_0002_0021.InfoData.AdsAddr <-> InfoData/AdsAddr
//     PlcTask Inputs/GVL_iXlinker.EtherCAT_Master_ERxxxx.Beckhoff_ER3xxx.Beckhoff_ER3xxxEK1122.A_0006_ER3184_0002_0021.InfoData.State <-> InfoData/State
//   PLC/PLC Instance <-> EtherCAT Master ERxxxx/Beckhoff ER3xxx/Beckhoff ER3xxxEK1122/A_0007(ER3184-1002-0020)
//     PlcTask Inputs/GVL_iXlinker.EtherCAT_Master_ERxxxx.Beckhoff_ER3xxx.Beckhoff_ER3xxxEK1122.A_0007_ER3184_1002_0020.AI_Standard_Channel_1.Status/Underrange <-> AI Standard Channel 1/Status/Underrange
//     PlcTask Inputs/GVL_iXlinker.EtherCAT_Master_ERxxxx.Beckhoff_ER3xxx.Beckhoff_ER3xxxEK1122.A_0007_ER3184_1002_0020.AI_Standard_Channel_2.Status/Underrange <-> AI Standard Channel 2/Status/Underrange
//     PlcTask Inputs/GVL_iXlinker.EtherCAT_Master_ERxxxx.Beckhoff_ER3xxx.Beckhoff_ER3xxxEK1122.A_0007_ER3184_1002_0020.AI_Standard_Channel_3.Status/Underrange <-> AI Standard Channel 3/Status/Underrange
//     PlcTask Inputs/GVL_iXlinker.EtherCAT_Master_ERxxxx.Beckhoff_ER3xxx.Beckhoff_ER3xxxEK1122.A_0007_ER3184_1002_0020.AI_Standard_Channel_4.Status/Underrange <-> AI Standard Channel 4/Status/Underrange
//     PlcTask Inputs/GVL_iXlinker.EtherCAT_Master_ERxxxx.Beckhoff_ER3xxx.Beckhoff_ER3xxxEK1122.A_0007_ER3184_1002_0020.AI_Standard_Channel_1.Status/Overrange <-> AI Standard Channel 1/Status/Overrange
//     PlcTask Inputs/GVL_iXlinker.EtherCAT_Master_ERxxxx.Beckhoff_ER3xxx.Beckhoff_ER3xxxEK1122.A_0007_ER3184_1002_0020.AI_Standard_Channel_2.Status/Overrange <-> AI Standard Channel 2/Status/Overrange
//     PlcTask Inputs/GVL_iXlinker.EtherCAT_Master_ERxxxx.Beckhoff_ER3xxx.Beckhoff_ER3xxxEK1122.A_0007_ER3184_1002_0020.AI_Standard_Channel_3.Status/Overrange <-> AI Standard Channel 3/Status/Overrange
//     PlcTask Inputs/GVL_iXlinker.EtherCAT_Master_ERxxxx.Beckhoff_ER3xxx.Beckhoff_ER3xxxEK1122.A_0007_ER3184_1002_0020.AI_Standard_Channel_4.Status/Overrange <-> AI Standard Channel 4/Status/Overrange
//     PlcTask Inputs/GVL_iXlinker.EtherCAT_Master_ERxxxx.Beckhoff_ER3xxx.Beckhoff_ER3xxxEK1122.A_0007_ER3184_1002_0020.AI_Standard_Channel_1.Status/Limit_1 <-> AI Standard Channel 1/Status/Limit 1
//     PlcTask Inputs/GVL_iXlinker.EtherCAT_Master_ERxxxx.Beckhoff_ER3xxx.Beckhoff_ER3xxxEK1122.A_0007_ER3184_1002_0020.AI_Standard_Channel_1.Status/Limit_2 <-> AI Standard Channel 1/Status/Limit 2
//     PlcTask Inputs/GVL_iXlinker.EtherCAT_Master_ERxxxx.Beckhoff_ER3xxx.Beckhoff_ER3xxxEK1122.A_0007_ER3184_1002_0020.AI_Standard_Channel_2.Status/Limit_1 <-> AI Standard Channel 2/Status/Limit 1
//     PlcTask Inputs/GVL_iXlinker.EtherCAT_Master_ERxxxx.Beckhoff_ER3xxx.Beckhoff_ER3xxxEK1122.A_0007_ER3184_1002_0020.AI_Standard_Channel_2.Status/Limit_2 <-> AI Standard Channel 2/Status/Limit 2
//     PlcTask Inputs/GVL_iXlinker.EtherCAT_Master_ERxxxx.Beckhoff_ER3xxx.Beckhoff_ER3xxxEK1122.A_0007_ER3184_1002_0020.AI_Standard_Channel_3.Status/Limit_1 <-> AI Standard Channel 3/Status/Limit 1
//     PlcTask Inputs/GVL_iXlinker.EtherCAT_Master_ERxxxx.Beckhoff_ER3xxx.Beckhoff_ER3xxxEK1122.A_0007_ER3184_1002_0020.AI_Standard_Channel_3.Status/Limit_2 <-> AI Standard Channel 3/Status/Limit 2
//     PlcTask Inputs/GVL_iXlinker.EtherCAT_Master_ERxxxx.Beckhoff_ER3xxx.Beckhoff_ER3xxxEK1122.A_0007_ER3184_1002_0020.AI_Standard_Channel_4.Status/Limit_1 <-> AI Standard Channel 4/Status/Limit 1
//     PlcTask Inputs/GVL_iXlinker.EtherCAT_Master_ERxxxx.Beckhoff_ER3xxx.Beckhoff_ER3xxxEK1122.A_0007_ER3184_1002_0020.AI_Standard_Channel_4.Status/Limit_2 <-> AI Standard Channel 4/Status/Limit 2
//     PlcTask Inputs/GVL_iXlinker.EtherCAT_Master_ERxxxx.Beckhoff_ER3xxx.Beckhoff_ER3xxxEK1122.A_0007_ER3184_1002_0020.AI_Standard_Channel_1.Status/Error <-> AI Standard Channel 1/Status/Error
//     PlcTask Inputs/GVL_iXlinker.EtherCAT_Master_ERxxxx.Beckhoff_ER3xxx.Beckhoff_ER3xxxEK1122.A_0007_ER3184_1002_0020.AI_Standard_Channel_2.Status/Error <-> AI Standard Channel 2/Status/Error
//     PlcTask Inputs/GVL_iXlinker.EtherCAT_Master_ERxxxx.Beckhoff_ER3xxx.Beckhoff_ER3xxxEK1122.A_0007_ER3184_1002_0020.AI_Standard_Channel_3.Status/Error <-> AI Standard Channel 3/Status/Error
//     PlcTask Inputs/GVL_iXlinker.EtherCAT_Master_ERxxxx.Beckhoff_ER3xxx.Beckhoff_ER3xxxEK1122.A_0007_ER3184_1002_0020.AI_Standard_Channel_4.Status/Error <-> AI Standard Channel 4/Status/Error
//     PlcTask Inputs/GVL_iXlinker.EtherCAT_Master_ERxxxx.Beckhoff_ER3xxx.Beckhoff_ER3xxxEK1122.A_0007_ER3184_1002_0020.AI_Standard_Channel_1.Status/Sync_error <-> AI Standard Channel 1/Status/Sync error
//     PlcTask Inputs/GVL_iXlinker.EtherCAT_Master_ERxxxx.Beckhoff_ER3xxx.Beckhoff_ER3xxxEK1122.A_0007_ER3184_1002_0020.AI_Standard_Channel_2.Status/Sync_error <-> AI Standard Channel 2/Status/Sync error
//     PlcTask Inputs/GVL_iXlinker.EtherCAT_Master_ERxxxx.Beckhoff_ER3xxx.Beckhoff_ER3xxxEK1122.A_0007_ER3184_1002_0020.AI_Standard_Channel_3.Status/Sync_error <-> AI Standard Channel 3/Status/Sync error
//     PlcTask Inputs/GVL_iXlinker.EtherCAT_Master_ERxxxx.Beckhoff_ER3xxx.Beckhoff_ER3xxxEK1122.A_0007_ER3184_1002_0020.AI_Standard_Channel_4.Status/Sync_error <-> AI Standard Channel 4/Status/Sync error
//     PlcTask Inputs/GVL_iXlinker.EtherCAT_Master_ERxxxx.Beckhoff_ER3xxx.Beckhoff_ER3xxxEK1122.A_0007_ER3184_1002_0020.AI_Standard_Channel_1.Status/TxPDO_State <-> AI Standard Channel 1/Status/TxPDO State
//     PlcTask Inputs/GVL_iXlinker.EtherCAT_Master_ERxxxx.Beckhoff_ER3xxx.Beckhoff_ER3xxxEK1122.A_0007_ER3184_1002_0020.AI_Standard_Channel_2.Status/TxPDO_State <-> AI Standard Channel 2/Status/TxPDO State
//     PlcTask Inputs/GVL_iXlinker.EtherCAT_Master_ERxxxx.Beckhoff_ER3xxx.Beckhoff_ER3xxxEK1122.A_0007_ER3184_1002_0020.AI_Standard_Channel_3.Status/TxPDO_State <-> AI Standard Channel 3/Status/TxPDO State
//     PlcTask Inputs/GVL_iXlinker.EtherCAT_Master_ERxxxx.Beckhoff_ER3xxx.Beckhoff_ER3xxxEK1122.A_0007_ER3184_1002_0020.AI_Standard_Channel_4.Status/TxPDO_State <-> AI Standard Channel 4/Status/TxPDO State
//     PlcTask Inputs/GVL_iXlinker.EtherCAT_Master_ERxxxx.Beckhoff_ER3xxx.Beckhoff_ER3xxxEK1122.A_0007_ER3184_1002_0020.AI_Standard_Channel_1.Status/TxPDO_Toggle <-> AI Standard Channel 1/Status/TxPDO Toggle
//     PlcTask Inputs/GVL_iXlinker.EtherCAT_Master_ERxxxx.Beckhoff_ER3xxx.Beckhoff_ER3xxxEK1122.A_0007_ER3184_1002_0020.AI_Standard_Channel_2.Status/TxPDO_Toggle <-> AI Standard Channel 2/Status/TxPDO Toggle
//     PlcTask Inputs/GVL_iXlinker.EtherCAT_Master_ERxxxx.Beckhoff_ER3xxx.Beckhoff_ER3xxxEK1122.A_0007_ER3184_1002_0020.AI_Standard_Channel_3.Status/TxPDO_Toggle <-> AI Standard Channel 3/Status/TxPDO Toggle
//     PlcTask Inputs/GVL_iXlinker.EtherCAT_Master_ERxxxx.Beckhoff_ER3xxx.Beckhoff_ER3xxxEK1122.A_0007_ER3184_1002_0020.AI_Standard_Channel_4.Status/TxPDO_Toggle <-> AI Standard Channel 4/Status/TxPDO Toggle
//     PlcTask Inputs/GVL_iXlinker.EtherCAT_Master_ERxxxx.Beckhoff_ER3xxx.Beckhoff_ER3xxxEK1122.A_0007_ER3184_1002_0020.AI_Standard_Channel_1.Value <-> AI Standard Channel 1/Value
//     PlcTask Inputs/GVL_iXlinker.EtherCAT_Master_ERxxxx.Beckhoff_ER3xxx.Beckhoff_ER3xxxEK1122.A_0007_ER3184_1002_0020.AI_Standard_Channel_2.Value <-> AI Standard Channel 2/Value
//     PlcTask Inputs/GVL_iXlinker.EtherCAT_Master_ERxxxx.Beckhoff_ER3xxx.Beckhoff_ER3xxxEK1122.A_0007_ER3184_1002_0020.AI_Standard_Channel_3.Value <-> AI Standard Channel 3/Value
//     PlcTask Inputs/GVL_iXlinker.EtherCAT_Master_ERxxxx.Beckhoff_ER3xxx.Beckhoff_ER3xxxEK1122.A_0007_ER3184_1002_0020.AI_Standard_Channel_4.Value <-> AI Standard Channel 4/Value
//     PlcTask Inputs/GVL_iXlinker.EtherCAT_Master_ERxxxx.Beckhoff_ER3xxx.Beckhoff_ER3xxxEK1122.A_0007_ER3184_1002_0020.WcState.WcState <-> WcState/WcState
//     PlcTask Inputs/GVL_iXlinker.EtherCAT_Master_ERxxxx.Beckhoff_ER3xxx.Beckhoff_ER3xxxEK1122.A_0007_ER3184_1002_0020.WcState.InputToggle <-> WcState/InputToggle
//     PlcTask Inputs/GVL_iXlinker.EtherCAT_Master_ERxxxx.Beckhoff_ER3xxx.Beckhoff_ER3xxxEK1122.A_0007_ER3184_1002_0020.InfoData.AdsAddr <-> InfoData/AdsAddr
//     PlcTask Inputs/GVL_iXlinker.EtherCAT_Master_ERxxxx.Beckhoff_ER3xxx.Beckhoff_ER3xxxEK1122.A_0007_ER3184_1002_0020.InfoData.State <-> InfoData/State
//   PLC/PLC Instance <-> EtherCAT Master ERxxxx/Beckhoff ER3xxx/Beckhoff ER3xxxEK1122/A_0008(ER3184-1002-0021)
//     PlcTask Inputs/GVL_iXlinker.EtherCAT_Master_ERxxxx.Beckhoff_ER3xxx.Beckhoff_ER3xxxEK1122.A_0008_ER3184_1002_0021.AI_Standard_Channel_1.Status/Underrange <-> AI Standard Channel 1/Status/Underrange
//     PlcTask Inputs/GVL_iXlinker.EtherCAT_Master_ERxxxx.Beckhoff_ER3xxx.Beckhoff_ER3xxxEK1122.A_0008_ER3184_1002_0021.AI_Standard_Channel_2.Status/Underrange <-> AI Standard Channel 2/Status/Underrange
//     PlcTask Inputs/GVL_iXlinker.EtherCAT_Master_ERxxxx.Beckhoff_ER3xxx.Beckhoff_ER3xxxEK1122.A_0008_ER3184_1002_0021.AI_Standard_Channel_3.Status/Underrange <-> AI Standard Channel 3/Status/Underrange
//     PlcTask Inputs/GVL_iXlinker.EtherCAT_Master_ERxxxx.Beckhoff_ER3xxx.Beckhoff_ER3xxxEK1122.A_0008_ER3184_1002_0021.AI_Standard_Channel_4.Status/Underrange <-> AI Standard Channel 4/Status/Underrange
//     PlcTask Inputs/GVL_iXlinker.EtherCAT_Master_ERxxxx.Beckhoff_ER3xxx.Beckhoff_ER3xxxEK1122.A_0008_ER3184_1002_0021.AI_Standard_Channel_1.Status/Overrange <-> AI Standard Channel 1/Status/Overrange
//     PlcTask Inputs/GVL_iXlinker.EtherCAT_Master_ERxxxx.Beckhoff_ER3xxx.Beckhoff_ER3xxxEK1122.A_0008_ER3184_1002_0021.AI_Standard_Channel_2.Status/Overrange <-> AI Standard Channel 2/Status/Overrange
//     PlcTask Inputs/GVL_iXlinker.EtherCAT_Master_ERxxxx.Beckhoff_ER3xxx.Beckhoff_ER3xxxEK1122.A_0008_ER3184_1002_0021.AI_Standard_Channel_3.Status/Overrange <-> AI Standard Channel 3/Status/Overrange
//     PlcTask Inputs/GVL_iXlinker.EtherCAT_Master_ERxxxx.Beckhoff_ER3xxx.Beckhoff_ER3xxxEK1122.A_0008_ER3184_1002_0021.AI_Standard_Channel_4.Status/Overrange <-> AI Standard Channel 4/Status/Overrange
//     PlcTask Inputs/GVL_iXlinker.EtherCAT_Master_ERxxxx.Beckhoff_ER3xxx.Beckhoff_ER3xxxEK1122.A_0008_ER3184_1002_0021.AI_Standard_Channel_1.Status/Limit_1 <-> AI Standard Channel 1/Status/Limit 1
//     PlcTask Inputs/GVL_iXlinker.EtherCAT_Master_ERxxxx.Beckhoff_ER3xxx.Beckhoff_ER3xxxEK1122.A_0008_ER3184_1002_0021.AI_Standard_Channel_1.Status/Limit_2 <-> AI Standard Channel 1/Status/Limit 2
//     PlcTask Inputs/GVL_iXlinker.EtherCAT_Master_ERxxxx.Beckhoff_ER3xxx.Beckhoff_ER3xxxEK1122.A_0008_ER3184_1002_0021.AI_Standard_Channel_2.Status/Limit_1 <-> AI Standard Channel 2/Status/Limit 1
//     PlcTask Inputs/GVL_iXlinker.EtherCAT_Master_ERxxxx.Beckhoff_ER3xxx.Beckhoff_ER3xxxEK1122.A_0008_ER3184_1002_0021.AI_Standard_Channel_2.Status/Limit_2 <-> AI Standard Channel 2/Status/Limit 2
//     PlcTask Inputs/GVL_iXlinker.EtherCAT_Master_ERxxxx.Beckhoff_ER3xxx.Beckhoff_ER3xxxEK1122.A_0008_ER3184_1002_0021.AI_Standard_Channel_3.Status/Limit_1 <-> AI Standard Channel 3/Status/Limit 1
//     PlcTask Inputs/GVL_iXlinker.EtherCAT_Master_ERxxxx.Beckhoff_ER3xxx.Beckhoff_ER3xxxEK1122.A_0008_ER3184_1002_0021.AI_Standard_Channel_3.Status/Limit_2 <-> AI Standard Channel 3/Status/Limit 2
//     PlcTask Inputs/GVL_iXlinker.EtherCAT_Master_ERxxxx.Beckhoff_ER3xxx.Beckhoff_ER3xxxEK1122.A_0008_ER3184_1002_0021.AI_Standard_Channel_4.Status/Limit_1 <-> AI Standard Channel 4/Status/Limit 1
//     PlcTask Inputs/GVL_iXlinker.EtherCAT_Master_ERxxxx.Beckhoff_ER3xxx.Beckhoff_ER3xxxEK1122.A_0008_ER3184_1002_0021.AI_Standard_Channel_4.Status/Limit_2 <-> AI Standard Channel 4/Status/Limit 2
//     PlcTask Inputs/GVL_iXlinker.EtherCAT_Master_ERxxxx.Beckhoff_ER3xxx.Beckhoff_ER3xxxEK1122.A_0008_ER3184_1002_0021.AI_Standard_Channel_1.Status/Error <-> AI Standard Channel 1/Status/Error
//     PlcTask Inputs/GVL_iXlinker.EtherCAT_Master_ERxxxx.Beckhoff_ER3xxx.Beckhoff_ER3xxxEK1122.A_0008_ER3184_1002_0021.AI_Standard_Channel_2.Status/Error <-> AI Standard Channel 2/Status/Error
//     PlcTask Inputs/GVL_iXlinker.EtherCAT_Master_ERxxxx.Beckhoff_ER3xxx.Beckhoff_ER3xxxEK1122.A_0008_ER3184_1002_0021.AI_Standard_Channel_3.Status/Error <-> AI Standard Channel 3/Status/Error
//     PlcTask Inputs/GVL_iXlinker.EtherCAT_Master_ERxxxx.Beckhoff_ER3xxx.Beckhoff_ER3xxxEK1122.A_0008_ER3184_1002_0021.AI_Standard_Channel_4.Status/Error <-> AI Standard Channel 4/Status/Error
//     PlcTask Inputs/GVL_iXlinker.EtherCAT_Master_ERxxxx.Beckhoff_ER3xxx.Beckhoff_ER3xxxEK1122.A_0008_ER3184_1002_0021.AI_Standard_Channel_1.Status/Sync_error <-> AI Standard Channel 1/Status/Sync error
//     PlcTask Inputs/GVL_iXlinker.EtherCAT_Master_ERxxxx.Beckhoff_ER3xxx.Beckhoff_ER3xxxEK1122.A_0008_ER3184_1002_0021.AI_Standard_Channel_2.Status/Sync_error <-> AI Standard Channel 2/Status/Sync error
//     PlcTask Inputs/GVL_iXlinker.EtherCAT_Master_ERxxxx.Beckhoff_ER3xxx.Beckhoff_ER3xxxEK1122.A_0008_ER3184_1002_0021.AI_Standard_Channel_3.Status/Sync_error <-> AI Standard Channel 3/Status/Sync error
//     PlcTask Inputs/GVL_iXlinker.EtherCAT_Master_ERxxxx.Beckhoff_ER3xxx.Beckhoff_ER3xxxEK1122.A_0008_ER3184_1002_0021.AI_Standard_Channel_4.Status/Sync_error <-> AI Standard Channel 4/Status/Sync error
//     PlcTask Inputs/GVL_iXlinker.EtherCAT_Master_ERxxxx.Beckhoff_ER3xxx.Beckhoff_ER3xxxEK1122.A_0008_ER3184_1002_0021.AI_Standard_Channel_1.Status/TxPDO_State <-> AI Standard Channel 1/Status/TxPDO State
//     PlcTask Inputs/GVL_iXlinker.EtherCAT_Master_ERxxxx.Beckhoff_ER3xxx.Beckhoff_ER3xxxEK1122.A_0008_ER3184_1002_0021.AI_Standard_Channel_2.Status/TxPDO_State <-> AI Standard Channel 2/Status/TxPDO State
//     PlcTask Inputs/GVL_iXlinker.EtherCAT_Master_ERxxxx.Beckhoff_ER3xxx.Beckhoff_ER3xxxEK1122.A_0008_ER3184_1002_0021.AI_Standard_Channel_3.Status/TxPDO_State <-> AI Standard Channel 3/Status/TxPDO State
//     PlcTask Inputs/GVL_iXlinker.EtherCAT_Master_ERxxxx.Beckhoff_ER3xxx.Beckhoff_ER3xxxEK1122.A_0008_ER3184_1002_0021.AI_Standard_Channel_4.Status/TxPDO_State <-> AI Standard Channel 4/Status/TxPDO State
//     PlcTask Inputs/GVL_iXlinker.EtherCAT_Master_ERxxxx.Beckhoff_ER3xxx.Beckhoff_ER3xxxEK1122.A_0008_ER3184_1002_0021.AI_Standard_Channel_1.Status/TxPDO_Toggle <-> AI Standard Channel 1/Status/TxPDO Toggle
//     PlcTask Inputs/GVL_iXlinker.EtherCAT_Master_ERxxxx.Beckhoff_ER3xxx.Beckhoff_ER3xxxEK1122.A_0008_ER3184_1002_0021.AI_Standard_Channel_2.Status/TxPDO_Toggle <-> AI Standard Channel 2/Status/TxPDO Toggle
//     PlcTask Inputs/GVL_iXlinker.EtherCAT_Master_ERxxxx.Beckhoff_ER3xxx.Beckhoff_ER3xxxEK1122.A_0008_ER3184_1002_0021.AI_Standard_Channel_3.Status/TxPDO_Toggle <-> AI Standard Channel 3/Status/TxPDO Toggle
//     PlcTask Inputs/GVL_iXlinker.EtherCAT_Master_ERxxxx.Beckhoff_ER3xxx.Beckhoff_ER3xxxEK1122.A_0008_ER3184_1002_0021.AI_Standard_Channel_4.Status/TxPDO_Toggle <-> AI Standard Channel 4/Status/TxPDO Toggle
//     PlcTask Inputs/GVL_iXlinker.EtherCAT_Master_ERxxxx.Beckhoff_ER3xxx.Beckhoff_ER3xxxEK1122.A_0008_ER3184_1002_0021.AI_Standard_Channel_1.Value <-> AI Standard Channel 1/Value
//     PlcTask Inputs/GVL_iXlinker.EtherCAT_Master_ERxxxx.Beckhoff_ER3xxx.Beckhoff_ER3xxxEK1122.A_0008_ER3184_1002_0021.AI_Standard_Channel_2.Value <-> AI Standard Channel 2/Value
//     PlcTask Inputs/GVL_iXlinker.EtherCAT_Master_ERxxxx.Beckhoff_ER3xxx.Beckhoff_ER3xxxEK1122.A_0008_ER3184_1002_0021.AI_Standard_Channel_3.Value <-> AI Standard Channel 3/Value
//     PlcTask Inputs/GVL_iXlinker.EtherCAT_Master_ERxxxx.Beckhoff_ER3xxx.Beckhoff_ER3xxxEK1122.A_0008_ER3184_1002_0021.AI_Standard_Channel_4.Value <-> AI Standard Channel 4/Value
//     PlcTask Inputs/GVL_iXlinker.EtherCAT_Master_ERxxxx.Beckhoff_ER3xxx.Beckhoff_ER3xxxEK1122.A_0008_ER3184_1002_0021.WcState.WcState <-> WcState/WcState
//     PlcTask Inputs/GVL_iXlinker.EtherCAT_Master_ERxxxx.Beckhoff_ER3xxx.Beckhoff_ER3xxxEK1122.A_0008_ER3184_1002_0021.WcState.InputToggle <-> WcState/InputToggle
//     PlcTask Inputs/GVL_iXlinker.EtherCAT_Master_ERxxxx.Beckhoff_ER3xxx.Beckhoff_ER3xxxEK1122.A_0008_ER3184_1002_0021.InfoData.AdsAddr <-> InfoData/AdsAddr
//     PlcTask Inputs/GVL_iXlinker.EtherCAT_Master_ERxxxx.Beckhoff_ER3xxx.Beckhoff_ER3xxxEK1122.A_0008_ER3184_1002_0021.InfoData.State <-> InfoData/State
//   PLC/PLC Instance <-> EtherCAT Master ERxxxx/Beckhoff ER3xxx/Beckhoff ER3xxxEK1122/A_0009(ER3204-0002-0016)
//     PlcTask Inputs/GVL_iXlinker.EtherCAT_Master_ERxxxx.Beckhoff_ER3xxx.Beckhoff_ER3xxxEK1122.A_0009_ER3204_0002_0016.RTD_RTDInputs_Channel_1.Status/Underrange <-> RTD RTDInputs Channel 1/Status/Underrange
//     PlcTask Inputs/GVL_iXlinker.EtherCAT_Master_ERxxxx.Beckhoff_ER3xxx.Beckhoff_ER3xxxEK1122.A_0009_ER3204_0002_0016.RTD_RTDInputs_Channel_2.Status/Underrange <-> RTD RTDInputs Channel 2/Status/Underrange
//     PlcTask Inputs/GVL_iXlinker.EtherCAT_Master_ERxxxx.Beckhoff_ER3xxx.Beckhoff_ER3xxxEK1122.A_0009_ER3204_0002_0016.RTD_RTDInputs_Channel_3.Status/Underrange <-> RTD RTDInputs Channel 3/Status/Underrange
//     PlcTask Inputs/GVL_iXlinker.EtherCAT_Master_ERxxxx.Beckhoff_ER3xxx.Beckhoff_ER3xxxEK1122.A_0009_ER3204_0002_0016.RTD_RTDInputs_Channel_4.Status/Underrange <-> RTD RTDInputs Channel 4/Status/Underrange
//     PlcTask Inputs/GVL_iXlinker.EtherCAT_Master_ERxxxx.Beckhoff_ER3xxx.Beckhoff_ER3xxxEK1122.A_0009_ER3204_0002_0016.RTD_RTDInputs_Channel_1.Status/Overrange <-> RTD RTDInputs Channel 1/Status/Overrange
//     PlcTask Inputs/GVL_iXlinker.EtherCAT_Master_ERxxxx.Beckhoff_ER3xxx.Beckhoff_ER3xxxEK1122.A_0009_ER3204_0002_0016.RTD_RTDInputs_Channel_2.Status/Overrange <-> RTD RTDInputs Channel 2/Status/Overrange
//     PlcTask Inputs/GVL_iXlinker.EtherCAT_Master_ERxxxx.Beckhoff_ER3xxx.Beckhoff_ER3xxxEK1122.A_0009_ER3204_0002_0016.RTD_RTDInputs_Channel_3.Status/Overrange <-> RTD RTDInputs Channel 3/Status/Overrange
//     PlcTask Inputs/GVL_iXlinker.EtherCAT_Master_ERxxxx.Beckhoff_ER3xxx.Beckhoff_ER3xxxEK1122.A_0009_ER3204_0002_0016.RTD_RTDInputs_Channel_4.Status/Overrange <-> RTD RTDInputs Channel 4/Status/Overrange
//     PlcTask Inputs/GVL_iXlinker.EtherCAT_Master_ERxxxx.Beckhoff_ER3xxx.Beckhoff_ER3xxxEK1122.A_0009_ER3204_0002_0016.RTD_RTDInputs_Channel_1.Status/Limit_1 <-> RTD RTDInputs Channel 1/Status/Limit 1
//     PlcTask Inputs/GVL_iXlinker.EtherCAT_Master_ERxxxx.Beckhoff_ER3xxx.Beckhoff_ER3xxxEK1122.A_0009_ER3204_0002_0016.RTD_RTDInputs_Channel_1.Status/Limit_2 <-> RTD RTDInputs Channel 1/Status/Limit 2
//     PlcTask Inputs/GVL_iXlinker.EtherCAT_Master_ERxxxx.Beckhoff_ER3xxx.Beckhoff_ER3xxxEK1122.A_0009_ER3204_0002_0016.RTD_RTDInputs_Channel_2.Status/Limit_1 <-> RTD RTDInputs Channel 2/Status/Limit 1
//     PlcTask Inputs/GVL_iXlinker.EtherCAT_Master_ERxxxx.Beckhoff_ER3xxx.Beckhoff_ER3xxxEK1122.A_0009_ER3204_0002_0016.RTD_RTDInputs_Channel_2.Status/Limit_2 <-> RTD RTDInputs Channel 2/Status/Limit 2
//     PlcTask Inputs/GVL_iXlinker.EtherCAT_Master_ERxxxx.Beckhoff_ER3xxx.Beckhoff_ER3xxxEK1122.A_0009_ER3204_0002_0016.RTD_RTDInputs_Channel_3.Status/Limit_1 <-> RTD RTDInputs Channel 3/Status/Limit 1
//     PlcTask Inputs/GVL_iXlinker.EtherCAT_Master_ERxxxx.Beckhoff_ER3xxx.Beckhoff_ER3xxxEK1122.A_0009_ER3204_0002_0016.RTD_RTDInputs_Channel_3.Status/Limit_2 <-> RTD RTDInputs Channel 3/Status/Limit 2
//     PlcTask Inputs/GVL_iXlinker.EtherCAT_Master_ERxxxx.Beckhoff_ER3xxx.Beckhoff_ER3xxxEK1122.A_0009_ER3204_0002_0016.RTD_RTDInputs_Channel_4.Status/Limit_1 <-> RTD RTDInputs Channel 4/Status/Limit 1
//     PlcTask Inputs/GVL_iXlinker.EtherCAT_Master_ERxxxx.Beckhoff_ER3xxx.Beckhoff_ER3xxxEK1122.A_0009_ER3204_0002_0016.RTD_RTDInputs_Channel_4.Status/Limit_2 <-> RTD RTDInputs Channel 4/Status/Limit 2
//     PlcTask Inputs/GVL_iXlinker.EtherCAT_Master_ERxxxx.Beckhoff_ER3xxx.Beckhoff_ER3xxxEK1122.A_0009_ER3204_0002_0016.RTD_RTDInputs_Channel_1.Status/Error <-> RTD RTDInputs Channel 1/Status/Error
//     PlcTask Inputs/GVL_iXlinker.EtherCAT_Master_ERxxxx.Beckhoff_ER3xxx.Beckhoff_ER3xxxEK1122.A_0009_ER3204_0002_0016.RTD_RTDInputs_Channel_2.Status/Error <-> RTD RTDInputs Channel 2/Status/Error
//     PlcTask Inputs/GVL_iXlinker.EtherCAT_Master_ERxxxx.Beckhoff_ER3xxx.Beckhoff_ER3xxxEK1122.A_0009_ER3204_0002_0016.RTD_RTDInputs_Channel_3.Status/Error <-> RTD RTDInputs Channel 3/Status/Error
//     PlcTask Inputs/GVL_iXlinker.EtherCAT_Master_ERxxxx.Beckhoff_ER3xxx.Beckhoff_ER3xxxEK1122.A_0009_ER3204_0002_0016.RTD_RTDInputs_Channel_4.Status/Error <-> RTD RTDInputs Channel 4/Status/Error
//     PlcTask Inputs/GVL_iXlinker.EtherCAT_Master_ERxxxx.Beckhoff_ER3xxx.Beckhoff_ER3xxxEK1122.A_0009_ER3204_0002_0016.RTD_RTDInputs_Channel_1.Status/Sync_error <-> RTD RTDInputs Channel 1/Status/Sync error
//     PlcTask Inputs/GVL_iXlinker.EtherCAT_Master_ERxxxx.Beckhoff_ER3xxx.Beckhoff_ER3xxxEK1122.A_0009_ER3204_0002_0016.RTD_RTDInputs_Channel_2.Status/Sync_error <-> RTD RTDInputs Channel 2/Status/Sync error
//     PlcTask Inputs/GVL_iXlinker.EtherCAT_Master_ERxxxx.Beckhoff_ER3xxx.Beckhoff_ER3xxxEK1122.A_0009_ER3204_0002_0016.RTD_RTDInputs_Channel_3.Status/Sync_error <-> RTD RTDInputs Channel 3/Status/Sync error
//     PlcTask Inputs/GVL_iXlinker.EtherCAT_Master_ERxxxx.Beckhoff_ER3xxx.Beckhoff_ER3xxxEK1122.A_0009_ER3204_0002_0016.RTD_RTDInputs_Channel_4.Status/Sync_error <-> RTD RTDInputs Channel 4/Status/Sync error
//     PlcTask Inputs/GVL_iXlinker.EtherCAT_Master_ERxxxx.Beckhoff_ER3xxx.Beckhoff_ER3xxxEK1122.A_0009_ER3204_0002_0016.RTD_RTDInputs_Channel_1.Status/TxPDO_State <-> RTD RTDInputs Channel 1/Status/TxPDO State
//     PlcTask Inputs/GVL_iXlinker.EtherCAT_Master_ERxxxx.Beckhoff_ER3xxx.Beckhoff_ER3xxxEK1122.A_0009_ER3204_0002_0016.RTD_RTDInputs_Channel_2.Status/TxPDO_State <-> RTD RTDInputs Channel 2/Status/TxPDO State
//     PlcTask Inputs/GVL_iXlinker.EtherCAT_Master_ERxxxx.Beckhoff_ER3xxx.Beckhoff_ER3xxxEK1122.A_0009_ER3204_0002_0016.RTD_RTDInputs_Channel_3.Status/TxPDO_State <-> RTD RTDInputs Channel 3/Status/TxPDO State
//     PlcTask Inputs/GVL_iXlinker.EtherCAT_Master_ERxxxx.Beckhoff_ER3xxx.Beckhoff_ER3xxxEK1122.A_0009_ER3204_0002_0016.RTD_RTDInputs_Channel_4.Status/TxPDO_State <-> RTD RTDInputs Channel 4/Status/TxPDO State
//     PlcTask Inputs/GVL_iXlinker.EtherCAT_Master_ERxxxx.Beckhoff_ER3xxx.Beckhoff_ER3xxxEK1122.A_0009_ER3204_0002_0016.RTD_RTDInputs_Channel_1.Status/TxPDO_Toggle <-> RTD RTDInputs Channel 1/Status/TxPDO Toggle
//     PlcTask Inputs/GVL_iXlinker.EtherCAT_Master_ERxxxx.Beckhoff_ER3xxx.Beckhoff_ER3xxxEK1122.A_0009_ER3204_0002_0016.RTD_RTDInputs_Channel_2.Status/TxPDO_Toggle <-> RTD RTDInputs Channel 2/Status/TxPDO Toggle
//     PlcTask Inputs/GVL_iXlinker.EtherCAT_Master_ERxxxx.Beckhoff_ER3xxx.Beckhoff_ER3xxxEK1122.A_0009_ER3204_0002_0016.RTD_RTDInputs_Channel_3.Status/TxPDO_Toggle <-> RTD RTDInputs Channel 3/Status/TxPDO Toggle
//     PlcTask Inputs/GVL_iXlinker.EtherCAT_Master_ERxxxx.Beckhoff_ER3xxx.Beckhoff_ER3xxxEK1122.A_0009_ER3204_0002_0016.RTD_RTDInputs_Channel_4.Status/TxPDO_Toggle <-> RTD RTDInputs Channel 4/Status/TxPDO Toggle
//     PlcTask Inputs/GVL_iXlinker.EtherCAT_Master_ERxxxx.Beckhoff_ER3xxx.Beckhoff_ER3xxxEK1122.A_0009_ER3204_0002_0016.RTD_RTDInputs_Channel_1.Value <-> RTD RTDInputs Channel 1/Value
//     PlcTask Inputs/GVL_iXlinker.EtherCAT_Master_ERxxxx.Beckhoff_ER3xxx.Beckhoff_ER3xxxEK1122.A_0009_ER3204_0002_0016.RTD_RTDInputs_Channel_2.Value <-> RTD RTDInputs Channel 2/Value
//     PlcTask Inputs/GVL_iXlinker.EtherCAT_Master_ERxxxx.Beckhoff_ER3xxx.Beckhoff_ER3xxxEK1122.A_0009_ER3204_0002_0016.RTD_RTDInputs_Channel_3.Value <-> RTD RTDInputs Channel 3/Value
//     PlcTask Inputs/GVL_iXlinker.EtherCAT_Master_ERxxxx.Beckhoff_ER3xxx.Beckhoff_ER3xxxEK1122.A_0009_ER3204_0002_0016.RTD_RTDInputs_Channel_4.Value <-> RTD RTDInputs Channel 4/Value
//     PlcTask Inputs/GVL_iXlinker.EtherCAT_Master_ERxxxx.Beckhoff_ER3xxx.Beckhoff_ER3xxxEK1122.A_0009_ER3204_0002_0016.WcState.WcState <-> WcState/WcState
//     PlcTask Inputs/GVL_iXlinker.EtherCAT_Master_ERxxxx.Beckhoff_ER3xxx.Beckhoff_ER3xxxEK1122.A_0009_ER3204_0002_0016.WcState.InputToggle <-> WcState/InputToggle
//     PlcTask Inputs/GVL_iXlinker.EtherCAT_Master_ERxxxx.Beckhoff_ER3xxx.Beckhoff_ER3xxxEK1122.A_0009_ER3204_0002_0016.InfoData.AdsAddr <-> InfoData/AdsAddr
//     PlcTask Inputs/GVL_iXlinker.EtherCAT_Master_ERxxxx.Beckhoff_ER3xxx.Beckhoff_ER3xxxEK1122.A_0009_ER3204_0002_0016.InfoData.State <-> InfoData/State
//   PLC/PLC Instance <-> EtherCAT Master ERxxxx/Beckhoff ER3xxx/Beckhoff ER3xxxEK1122/A_0010(ER3204-0002-0020)
//     PlcTask Inputs/GVL_iXlinker.EtherCAT_Master_ERxxxx.Beckhoff_ER3xxx.Beckhoff_ER3xxxEK1122.A_0010_ER3204_0002_0020.RTD_RTDInputs_Channel_1.Status/Underrange <-> RTD RTDInputs Channel 1/Status/Underrange
//     PlcTask Inputs/GVL_iXlinker.EtherCAT_Master_ERxxxx.Beckhoff_ER3xxx.Beckhoff_ER3xxxEK1122.A_0010_ER3204_0002_0020.RTD_RTDInputs_Channel_2.Status/Underrange <-> RTD RTDInputs Channel 2/Status/Underrange
//     PlcTask Inputs/GVL_iXlinker.EtherCAT_Master_ERxxxx.Beckhoff_ER3xxx.Beckhoff_ER3xxxEK1122.A_0010_ER3204_0002_0020.RTD_RTDInputs_Channel_3.Status/Underrange <-> RTD RTDInputs Channel 3/Status/Underrange
//     PlcTask Inputs/GVL_iXlinker.EtherCAT_Master_ERxxxx.Beckhoff_ER3xxx.Beckhoff_ER3xxxEK1122.A_0010_ER3204_0002_0020.RTD_RTDInputs_Channel_4.Status/Underrange <-> RTD RTDInputs Channel 4/Status/Underrange
//     PlcTask Inputs/GVL_iXlinker.EtherCAT_Master_ERxxxx.Beckhoff_ER3xxx.Beckhoff_ER3xxxEK1122.A_0010_ER3204_0002_0020.RTD_RTDInputs_Channel_1.Status/Overrange <-> RTD RTDInputs Channel 1/Status/Overrange
//     PlcTask Inputs/GVL_iXlinker.EtherCAT_Master_ERxxxx.Beckhoff_ER3xxx.Beckhoff_ER3xxxEK1122.A_0010_ER3204_0002_0020.RTD_RTDInputs_Channel_2.Status/Overrange <-> RTD RTDInputs Channel 2/Status/Overrange
//     PlcTask Inputs/GVL_iXlinker.EtherCAT_Master_ERxxxx.Beckhoff_ER3xxx.Beckhoff_ER3xxxEK1122.A_0010_ER3204_0002_0020.RTD_RTDInputs_Channel_3.Status/Overrange <-> RTD RTDInputs Channel 3/Status/Overrange
//     PlcTask Inputs/GVL_iXlinker.EtherCAT_Master_ERxxxx.Beckhoff_ER3xxx.Beckhoff_ER3xxxEK1122.A_0010_ER3204_0002_0020.RTD_RTDInputs_Channel_4.Status/Overrange <-> RTD RTDInputs Channel 4/Status/Overrange
//     PlcTask Inputs/GVL_iXlinker.EtherCAT_Master_ERxxxx.Beckhoff_ER3xxx.Beckhoff_ER3xxxEK1122.A_0010_ER3204_0002_0020.RTD_RTDInputs_Channel_1.Status/Limit_1 <-> RTD RTDInputs Channel 1/Status/Limit 1
//     PlcTask Inputs/GVL_iXlinker.EtherCAT_Master_ERxxxx.Beckhoff_ER3xxx.Beckhoff_ER3xxxEK1122.A_0010_ER3204_0002_0020.RTD_RTDInputs_Channel_1.Status/Limit_2 <-> RTD RTDInputs Channel 1/Status/Limit 2
//     PlcTask Inputs/GVL_iXlinker.EtherCAT_Master_ERxxxx.Beckhoff_ER3xxx.Beckhoff_ER3xxxEK1122.A_0010_ER3204_0002_0020.RTD_RTDInputs_Channel_2.Status/Limit_1 <-> RTD RTDInputs Channel 2/Status/Limit 1
//     PlcTask Inputs/GVL_iXlinker.EtherCAT_Master_ERxxxx.Beckhoff_ER3xxx.Beckhoff_ER3xxxEK1122.A_0010_ER3204_0002_0020.RTD_RTDInputs_Channel_2.Status/Limit_2 <-> RTD RTDInputs Channel 2/Status/Limit 2
//     PlcTask Inputs/GVL_iXlinker.EtherCAT_Master_ERxxxx.Beckhoff_ER3xxx.Beckhoff_ER3xxxEK1122.A_0010_ER3204_0002_0020.RTD_RTDInputs_Channel_3.Status/Limit_1 <-> RTD RTDInputs Channel 3/Status/Limit 1
//     PlcTask Inputs/GVL_iXlinker.EtherCAT_Master_ERxxxx.Beckhoff_ER3xxx.Beckhoff_ER3xxxEK1122.A_0010_ER3204_0002_0020.RTD_RTDInputs_Channel_3.Status/Limit_2 <-> RTD RTDInputs Channel 3/Status/Limit 2
//     PlcTask Inputs/GVL_iXlinker.EtherCAT_Master_ERxxxx.Beckhoff_ER3xxx.Beckhoff_ER3xxxEK1122.A_0010_ER3204_0002_0020.RTD_RTDInputs_Channel_4.Status/Limit_1 <-> RTD RTDInputs Channel 4/Status/Limit 1
//     PlcTask Inputs/GVL_iXlinker.EtherCAT_Master_ERxxxx.Beckhoff_ER3xxx.Beckhoff_ER3xxxEK1122.A_0010_ER3204_0002_0020.RTD_RTDInputs_Channel_4.Status/Limit_2 <-> RTD RTDInputs Channel 4/Status/Limit 2
//     PlcTask Inputs/GVL_iXlinker.EtherCAT_Master_ERxxxx.Beckhoff_ER3xxx.Beckhoff_ER3xxxEK1122.A_0010_ER3204_0002_0020.RTD_RTDInputs_Channel_1.Status/Error <-> RTD RTDInputs Channel 1/Status/Error
//     PlcTask Inputs/GVL_iXlinker.EtherCAT_Master_ERxxxx.Beckhoff_ER3xxx.Beckhoff_ER3xxxEK1122.A_0010_ER3204_0002_0020.RTD_RTDInputs_Channel_2.Status/Error <-> RTD RTDInputs Channel 2/Status/Error
//     PlcTask Inputs/GVL_iXlinker.EtherCAT_Master_ERxxxx.Beckhoff_ER3xxx.Beckhoff_ER3xxxEK1122.A_0010_ER3204_0002_0020.RTD_RTDInputs_Channel_3.Status/Error <-> RTD RTDInputs Channel 3/Status/Error
//     PlcTask Inputs/GVL_iXlinker.EtherCAT_Master_ERxxxx.Beckhoff_ER3xxx.Beckhoff_ER3xxxEK1122.A_0010_ER3204_0002_0020.RTD_RTDInputs_Channel_4.Status/Error <-> RTD RTDInputs Channel 4/Status/Error
//     PlcTask Inputs/GVL_iXlinker.EtherCAT_Master_ERxxxx.Beckhoff_ER3xxx.Beckhoff_ER3xxxEK1122.A_0010_ER3204_0002_0020.RTD_RTDInputs_Channel_1.Status/Sync_error <-> RTD RTDInputs Channel 1/Status/Sync error
//     PlcTask Inputs/GVL_iXlinker.EtherCAT_Master_ERxxxx.Beckhoff_ER3xxx.Beckhoff_ER3xxxEK1122.A_0010_ER3204_0002_0020.RTD_RTDInputs_Channel_2.Status/Sync_error <-> RTD RTDInputs Channel 2/Status/Sync error
//     PlcTask Inputs/GVL_iXlinker.EtherCAT_Master_ERxxxx.Beckhoff_ER3xxx.Beckhoff_ER3xxxEK1122.A_0010_ER3204_0002_0020.RTD_RTDInputs_Channel_3.Status/Sync_error <-> RTD RTDInputs Channel 3/Status/Sync error
//     PlcTask Inputs/GVL_iXlinker.EtherCAT_Master_ERxxxx.Beckhoff_ER3xxx.Beckhoff_ER3xxxEK1122.A_0010_ER3204_0002_0020.RTD_RTDInputs_Channel_4.Status/Sync_error <-> RTD RTDInputs Channel 4/Status/Sync error
//     PlcTask Inputs/GVL_iXlinker.EtherCAT_Master_ERxxxx.Beckhoff_ER3xxx.Beckhoff_ER3xxxEK1122.A_0010_ER3204_0002_0020.RTD_RTDInputs_Channel_1.Status/TxPDO_State <-> RTD RTDInputs Channel 1/Status/TxPDO State
//     PlcTask Inputs/GVL_iXlinker.EtherCAT_Master_ERxxxx.Beckhoff_ER3xxx.Beckhoff_ER3xxxEK1122.A_0010_ER3204_0002_0020.RTD_RTDInputs_Channel_2.Status/TxPDO_State <-> RTD RTDInputs Channel 2/Status/TxPDO State
//     PlcTask Inputs/GVL_iXlinker.EtherCAT_Master_ERxxxx.Beckhoff_ER3xxx.Beckhoff_ER3xxxEK1122.A_0010_ER3204_0002_0020.RTD_RTDInputs_Channel_3.Status/TxPDO_State <-> RTD RTDInputs Channel 3/Status/TxPDO State
//     PlcTask Inputs/GVL_iXlinker.EtherCAT_Master_ERxxxx.Beckhoff_ER3xxx.Beckhoff_ER3xxxEK1122.A_0010_ER3204_0002_0020.RTD_RTDInputs_Channel_4.Status/TxPDO_State <-> RTD RTDInputs Channel 4/Status/TxPDO State
//     PlcTask Inputs/GVL_iXlinker.EtherCAT_Master_ERxxxx.Beckhoff_ER3xxx.Beckhoff_ER3xxxEK1122.A_0010_ER3204_0002_0020.RTD_RTDInputs_Channel_1.Status/TxPDO_Toggle <-> RTD RTDInputs Channel 1/Status/TxPDO Toggle
//     PlcTask Inputs/GVL_iXlinker.EtherCAT_Master_ERxxxx.Beckhoff_ER3xxx.Beckhoff_ER3xxxEK1122.A_0010_ER3204_0002_0020.RTD_RTDInputs_Channel_2.Status/TxPDO_Toggle <-> RTD RTDInputs Channel 2/Status/TxPDO Toggle
//     PlcTask Inputs/GVL_iXlinker.EtherCAT_Master_ERxxxx.Beckhoff_ER3xxx.Beckhoff_ER3xxxEK1122.A_0010_ER3204_0002_0020.RTD_RTDInputs_Channel_3.Status/TxPDO_Toggle <-> RTD RTDInputs Channel 3/Status/TxPDO Toggle
//     PlcTask Inputs/GVL_iXlinker.EtherCAT_Master_ERxxxx.Beckhoff_ER3xxx.Beckhoff_ER3xxxEK1122.A_0010_ER3204_0002_0020.RTD_RTDInputs_Channel_4.Status/TxPDO_Toggle <-> RTD RTDInputs Channel 4/Status/TxPDO Toggle
//     PlcTask Inputs/GVL_iXlinker.EtherCAT_Master_ERxxxx.Beckhoff_ER3xxx.Beckhoff_ER3xxxEK1122.A_0010_ER3204_0002_0020.RTD_RTDInputs_Channel_1.Value <-> RTD RTDInputs Channel 1/Value
//     PlcTask Inputs/GVL_iXlinker.EtherCAT_Master_ERxxxx.Beckhoff_ER3xxx.Beckhoff_ER3xxxEK1122.A_0010_ER3204_0002_0020.RTD_RTDInputs_Channel_2.Value <-> RTD RTDInputs Channel 2/Value
//     PlcTask Inputs/GVL_iXlinker.EtherCAT_Master_ERxxxx.Beckhoff_ER3xxx.Beckhoff_ER3xxxEK1122.A_0010_ER3204_0002_0020.RTD_RTDInputs_Channel_3.Value <-> RTD RTDInputs Channel 3/Value
//     PlcTask Inputs/GVL_iXlinker.EtherCAT_Master_ERxxxx.Beckhoff_ER3xxx.Beckhoff_ER3xxxEK1122.A_0010_ER3204_0002_0020.RTD_RTDInputs_Channel_4.Value <-> RTD RTDInputs Channel 4/Value
//     PlcTask Inputs/GVL_iXlinker.EtherCAT_Master_ERxxxx.Beckhoff_ER3xxx.Beckhoff_ER3xxxEK1122.A_0010_ER3204_0002_0020.WcState.WcState <-> WcState/WcState
//     PlcTask Inputs/GVL_iXlinker.EtherCAT_Master_ERxxxx.Beckhoff_ER3xxx.Beckhoff_ER3xxxEK1122.A_0010_ER3204_0002_0020.WcState.InputToggle <-> WcState/InputToggle
//     PlcTask Inputs/GVL_iXlinker.EtherCAT_Master_ERxxxx.Beckhoff_ER3xxx.Beckhoff_ER3xxxEK1122.A_0010_ER3204_0002_0020.InfoData.AdsAddr <-> InfoData/AdsAddr
//     PlcTask Inputs/GVL_iXlinker.EtherCAT_Master_ERxxxx.Beckhoff_ER3xxx.Beckhoff_ER3xxxEK1122.A_0010_ER3204_0002_0020.InfoData.State <-> InfoData/State
//   PLC/PLC Instance <-> EtherCAT Master ERxxxx/Beckhoff ER3xxx/Beckhoff ER3xxxEK1122/A_0011(ER3204-0002-0021)
//     PlcTask Inputs/GVL_iXlinker.EtherCAT_Master_ERxxxx.Beckhoff_ER3xxx.Beckhoff_ER3xxxEK1122.A_0011_ER3204_0002_0021.RTD_RTDInputs_Channel_1.Status/Underrange <-> RTD RTDInputs Channel 1/Status/Underrange
//     PlcTask Inputs/GVL_iXlinker.EtherCAT_Master_ERxxxx.Beckhoff_ER3xxx.Beckhoff_ER3xxxEK1122.A_0011_ER3204_0002_0021.RTD_RTDInputs_Channel_2.Status/Underrange <-> RTD RTDInputs Channel 2/Status/Underrange
//     PlcTask Inputs/GVL_iXlinker.EtherCAT_Master_ERxxxx.Beckhoff_ER3xxx.Beckhoff_ER3xxxEK1122.A_0011_ER3204_0002_0021.RTD_RTDInputs_Channel_3.Status/Underrange <-> RTD RTDInputs Channel 3/Status/Underrange
//     PlcTask Inputs/GVL_iXlinker.EtherCAT_Master_ERxxxx.Beckhoff_ER3xxx.Beckhoff_ER3xxxEK1122.A_0011_ER3204_0002_0021.RTD_RTDInputs_Channel_4.Status/Underrange <-> RTD RTDInputs Channel 4/Status/Underrange
//     PlcTask Inputs/GVL_iXlinker.EtherCAT_Master_ERxxxx.Beckhoff_ER3xxx.Beckhoff_ER3xxxEK1122.A_0011_ER3204_0002_0021.RTD_RTDInputs_Channel_1.Status/Overrange <-> RTD RTDInputs Channel 1/Status/Overrange
//     PlcTask Inputs/GVL_iXlinker.EtherCAT_Master_ERxxxx.Beckhoff_ER3xxx.Beckhoff_ER3xxxEK1122.A_0011_ER3204_0002_0021.RTD_RTDInputs_Channel_2.Status/Overrange <-> RTD RTDInputs Channel 2/Status/Overrange
//     PlcTask Inputs/GVL_iXlinker.EtherCAT_Master_ERxxxx.Beckhoff_ER3xxx.Beckhoff_ER3xxxEK1122.A_0011_ER3204_0002_0021.RTD_RTDInputs_Channel_3.Status/Overrange <-> RTD RTDInputs Channel 3/Status/Overrange
//     PlcTask Inputs/GVL_iXlinker.EtherCAT_Master_ERxxxx.Beckhoff_ER3xxx.Beckhoff_ER3xxxEK1122.A_0011_ER3204_0002_0021.RTD_RTDInputs_Channel_4.Status/Overrange <-> RTD RTDInputs Channel 4/Status/Overrange
//     PlcTask Inputs/GVL_iXlinker.EtherCAT_Master_ERxxxx.Beckhoff_ER3xxx.Beckhoff_ER3xxxEK1122.A_0011_ER3204_0002_0021.RTD_RTDInputs_Channel_1.Status/Limit_1 <-> RTD RTDInputs Channel 1/Status/Limit 1
//     PlcTask Inputs/GVL_iXlinker.EtherCAT_Master_ERxxxx.Beckhoff_ER3xxx.Beckhoff_ER3xxxEK1122.A_0011_ER3204_0002_0021.RTD_RTDInputs_Channel_1.Status/Limit_2 <-> RTD RTDInputs Channel 1/Status/Limit 2
//     PlcTask Inputs/GVL_iXlinker.EtherCAT_Master_ERxxxx.Beckhoff_ER3xxx.Beckhoff_ER3xxxEK1122.A_0011_ER3204_0002_0021.RTD_RTDInputs_Channel_2.Status/Limit_1 <-> RTD RTDInputs Channel 2/Status/Limit 1
//     PlcTask Inputs/GVL_iXlinker.EtherCAT_Master_ERxxxx.Beckhoff_ER3xxx.Beckhoff_ER3xxxEK1122.A_0011_ER3204_0002_0021.RTD_RTDInputs_Channel_2.Status/Limit_2 <-> RTD RTDInputs Channel 2/Status/Limit 2
//     PlcTask Inputs/GVL_iXlinker.EtherCAT_Master_ERxxxx.Beckhoff_ER3xxx.Beckhoff_ER3xxxEK1122.A_0011_ER3204_0002_0021.RTD_RTDInputs_Channel_3.Status/Limit_1 <-> RTD RTDInputs Channel 3/Status/Limit 1
//     PlcTask Inputs/GVL_iXlinker.EtherCAT_Master_ERxxxx.Beckhoff_ER3xxx.Beckhoff_ER3xxxEK1122.A_0011_ER3204_0002_0021.RTD_RTDInputs_Channel_3.Status/Limit_2 <-> RTD RTDInputs Channel 3/Status/Limit 2
//     PlcTask Inputs/GVL_iXlinker.EtherCAT_Master_ERxxxx.Beckhoff_ER3xxx.Beckhoff_ER3xxxEK1122.A_0011_ER3204_0002_0021.RTD_RTDInputs_Channel_4.Status/Limit_1 <-> RTD RTDInputs Channel 4/Status/Limit 1
//     PlcTask Inputs/GVL_iXlinker.EtherCAT_Master_ERxxxx.Beckhoff_ER3xxx.Beckhoff_ER3xxxEK1122.A_0011_ER3204_0002_0021.RTD_RTDInputs_Channel_4.Status/Limit_2 <-> RTD RTDInputs Channel 4/Status/Limit 2
//     PlcTask Inputs/GVL_iXlinker.EtherCAT_Master_ERxxxx.Beckhoff_ER3xxx.Beckhoff_ER3xxxEK1122.A_0011_ER3204_0002_0021.RTD_RTDInputs_Channel_1.Status/Error <-> RTD RTDInputs Channel 1/Status/Error
//     PlcTask Inputs/GVL_iXlinker.EtherCAT_Master_ERxxxx.Beckhoff_ER3xxx.Beckhoff_ER3xxxEK1122.A_0011_ER3204_0002_0021.RTD_RTDInputs_Channel_2.Status/Error <-> RTD RTDInputs Channel 2/Status/Error
//     PlcTask Inputs/GVL_iXlinker.EtherCAT_Master_ERxxxx.Beckhoff_ER3xxx.Beckhoff_ER3xxxEK1122.A_0011_ER3204_0002_0021.RTD_RTDInputs_Channel_3.Status/Error <-> RTD RTDInputs Channel 3/Status/Error
//     PlcTask Inputs/GVL_iXlinker.EtherCAT_Master_ERxxxx.Beckhoff_ER3xxx.Beckhoff_ER3xxxEK1122.A_0011_ER3204_0002_0021.RTD_RTDInputs_Channel_4.Status/Error <-> RTD RTDInputs Channel 4/Status/Error
//     PlcTask Inputs/GVL_iXlinker.EtherCAT_Master_ERxxxx.Beckhoff_ER3xxx.Beckhoff_ER3xxxEK1122.A_0011_ER3204_0002_0021.RTD_RTDInputs_Channel_1.Status/TxPDO_State <-> RTD RTDInputs Channel 1/Status/TxPDO State
//     PlcTask Inputs/GVL_iXlinker.EtherCAT_Master_ERxxxx.Beckhoff_ER3xxx.Beckhoff_ER3xxxEK1122.A_0011_ER3204_0002_0021.RTD_RTDInputs_Channel_2.Status/TxPDO_State <-> RTD RTDInputs Channel 2/Status/TxPDO State
//     PlcTask Inputs/GVL_iXlinker.EtherCAT_Master_ERxxxx.Beckhoff_ER3xxx.Beckhoff_ER3xxxEK1122.A_0011_ER3204_0002_0021.RTD_RTDInputs_Channel_3.Status/TxPDO_State <-> RTD RTDInputs Channel 3/Status/TxPDO State
//     PlcTask Inputs/GVL_iXlinker.EtherCAT_Master_ERxxxx.Beckhoff_ER3xxx.Beckhoff_ER3xxxEK1122.A_0011_ER3204_0002_0021.RTD_RTDInputs_Channel_4.Status/TxPDO_State <-> RTD RTDInputs Channel 4/Status/TxPDO State
//     PlcTask Inputs/GVL_iXlinker.EtherCAT_Master_ERxxxx.Beckhoff_ER3xxx.Beckhoff_ER3xxxEK1122.A_0011_ER3204_0002_0021.RTD_RTDInputs_Channel_1.Status/TxPDO_Toggle <-> RTD RTDInputs Channel 1/Status/TxPDO Toggle
//     PlcTask Inputs/GVL_iXlinker.EtherCAT_Master_ERxxxx.Beckhoff_ER3xxx.Beckhoff_ER3xxxEK1122.A_0011_ER3204_0002_0021.RTD_RTDInputs_Channel_2.Status/TxPDO_Toggle <-> RTD RTDInputs Channel 2/Status/TxPDO Toggle
//     PlcTask Inputs/GVL_iXlinker.EtherCAT_Master_ERxxxx.Beckhoff_ER3xxx.Beckhoff_ER3xxxEK1122.A_0011_ER3204_0002_0021.RTD_RTDInputs_Channel_3.Status/TxPDO_Toggle <-> RTD RTDInputs Channel 3/Status/TxPDO Toggle
//     PlcTask Inputs/GVL_iXlinker.EtherCAT_Master_ERxxxx.Beckhoff_ER3xxx.Beckhoff_ER3xxxEK1122.A_0011_ER3204_0002_0021.RTD_RTDInputs_Channel_4.Status/TxPDO_Toggle <-> RTD RTDInputs Channel 4/Status/TxPDO Toggle
//     PlcTask Inputs/GVL_iXlinker.EtherCAT_Master_ERxxxx.Beckhoff_ER3xxx.Beckhoff_ER3xxxEK1122.A_0011_ER3204_0002_0021.RTD_RTDInputs_Channel_1.Value <-> RTD RTDInputs Channel 1/Value
//     PlcTask Inputs/GVL_iXlinker.EtherCAT_Master_ERxxxx.Beckhoff_ER3xxx.Beckhoff_ER3xxxEK1122.A_0011_ER3204_0002_0021.RTD_RTDInputs_Channel_2.Value <-> RTD RTDInputs Channel 2/Value
//     PlcTask Inputs/GVL_iXlinker.EtherCAT_Master_ERxxxx.Beckhoff_ER3xxx.Beckhoff_ER3xxxEK1122.A_0011_ER3204_0002_0021.RTD_RTDInputs_Channel_3.Value <-> RTD RTDInputs Channel 3/Value
//     PlcTask Inputs/GVL_iXlinker.EtherCAT_Master_ERxxxx.Beckhoff_ER3xxx.Beckhoff_ER3xxxEK1122.A_0011_ER3204_0002_0021.RTD_RTDInputs_Channel_4.Value <-> RTD RTDInputs Channel 4/Value
//     PlcTask Inputs/GVL_iXlinker.EtherCAT_Master_ERxxxx.Beckhoff_ER3xxx.Beckhoff_ER3xxxEK1122.A_0011_ER3204_0002_0021.WcState.WcState <-> WcState/WcState
//     PlcTask Inputs/GVL_iXlinker.EtherCAT_Master_ERxxxx.Beckhoff_ER3xxx.Beckhoff_ER3xxxEK1122.A_0011_ER3204_0002_0021.WcState.InputToggle <-> WcState/InputToggle
//     PlcTask Inputs/GVL_iXlinker.EtherCAT_Master_ERxxxx.Beckhoff_ER3xxx.Beckhoff_ER3xxxEK1122.A_0011_ER3204_0002_0021.InfoData.AdsAddr <-> InfoData/AdsAddr
//     PlcTask Inputs/GVL_iXlinker.EtherCAT_Master_ERxxxx.Beckhoff_ER3xxx.Beckhoff_ER3xxxEK1122.A_0011_ER3204_0002_0021.InfoData.State <-> InfoData/State
//   PLC/PLC Instance <-> EtherCAT Master ERxxxx/Beckhoff ER3xxx/Beckhoff ER3xxxEK1122/A_0012(ER3314-0002-0021)
